Omron CX-Programmer project 新工程 (CX-Programmer 9.72)

# PLC 新PLC1: CJ1M CPU13
I/O table (CPU CJ1M-CPU13): rack 0 slot 0 CJ1W-SCU41-V1; rack 0 slot 1 CJ1W-DRM21; rack 0 slot 2 CJ1W-IA111; rack 0 slot 3 CJ1W-IA111; rack 0 slot 4 CJ1W-IA111; rack 0 slot 5 CJ1W-IA111; rack 0 slot 6 CJ1W-IA111; rack 0 slot 7 CJ1W-IA111; rack 0 slot 8 CJ1W-IA111; rack 0 slot 9 CJ1W-OC211; rack 1 slot 0 CJ1W-OC211; rack 1 slot 1 CJ1W-OC211; rack 1 slot 2 CJ1W-OC211; rack 1 slot 3 CJ1W-OC211; rack 1 slot 4 CJ1W-ID211; rack 1 slot 5 CJ1W-IA111; rack 1 slot 6 CJ1W-AD041-V1

## Global symbols (name address type ; comment)
0.00 BOOL  ; 右前按钮站闭点并
0.01 BOOL  ; 右前按钮站闭点串
0.02 BOOL  ; 右前按钮站开点串
0.04 BOOL  ; 左后按钮站闭点并
0.05 BOOL  ; 左后按钮站闭点串
0.06 BOOL  ; 左后按钮站开点串
150 CHANNEL  ; 1-16通道比较后的结果字
151 CHANNEL  ; 17-32通道比较后的结果字
2008.01 BOOL  ; RUN mode
2008.02 BOOL  ; 电子凸轮模块故障
2008.04 BOOL  ; Memory load completed
2008.06 BOOL  ; Memory load enable
30.00 BOOL  ; 高油压
30.01 BOOL  ; 1#高油压
30.03 BOOL  ; 主润滑次数正常
30.06 BOOL  ; 气垫润滑高压
30.07 BOOL  ; 油箱加热
30.08 BOOL  ; 润滑次数正常
30.09 BOOL  ; 低油压
30.13 BOOL  ; 主润滑次数正常
30.14 BOOL  ; 润滑正常
310.03 BOOL  ; 1#MB前开出停止
315.01 BOOL  ; 高油位
315.02 BOOL  ; 低油位
315.03 BOOL  ; 1#过滤器堵塞
315.04 BOOL  ; 2#过滤器堵塞
315.05 BOOL  ; 3#滤油器堵塞
315.06 BOOL  ; 高油压
315.07 BOOL  ; 低油压
316.00 BOOL  ; 模具更换
316.01 BOOL  ; 上死点300-0
316.02 BOOL  ; 数据编辑断
316.03 BOOL  ; 气垫落到底
316.06 BOOL  ; MB右开进停止
316.07 BOOL  ; 选择夹紧
316.08 BOOL  ; 选择放松
316.09 BOOL  ; MB落下（前）
316.10 BOOL  ; MB落下（后）
316.11 BOOL  ; MB夹紧压力
316.12 BOOL  ; MB放松压力
318.00 BOOL  ; 变频器正常
318.01 BOOL  ; 变频器电源合上
318.02 BOOL  ; 点动
318.03 BOOL  ; 单动
318.04 BOOL  ; 自动
318.05 BOOL  ; 安全栓复位
319.00 BOOL  ; 双阀故障
319.02 BOOL  ; 安全栓未就位
319.03 BOOL  ; 急停故障
319.04 BOOL  ; 工作台变频器正常
31.13 BOOL  ; 故障复位
31.14 BOOL  ; 急停防粘
31.15 BOOL  ; 紧急停止
320.02 BOOL  ; 润滑电机开关触点
320.04 BOOL  ; 电柜冷却开关触点
320.05 BOOL  ; 润滑电机停止
320.06 BOOL  ; 润滑电机开动
320.09 BOOL  ; 油箱加热开关触点
320.10 BOOL  ; 油箱温度正常
320.11 BOOL  ; 油箱加热停
320.12 BOOL  ; 油箱加热开
320.14 BOOL  ; 润滑电机运行
320.15 BOOL  ; 油箱加热
321.00 BOOL  ; 润滑正常
321.01 BOOL  ; 主电机温度正常
321.02 BOOL  ; 梯子限位
321.03 BOOL  ; 主电机热过载
321.04 BOOL  ; 主电机零速
321.10 BOOL  ; 主电机停止按钮
321.11 BOOL  ; 主电机启动按钮
321.12 BOOL  ; 飞轮制动限位1#
321.13 BOOL  ; 飞轮制动限位2#
321.15 BOOL  ; 主电机启动OK
322.00 BOOL  ; 主电机运行
322.10 BOOL  ; 数据编辑通/断
322.11 BOOL  ; 安全栓到位
322.13 BOOL  ; 液压保护过载
322.14 BOOL  ; 液压保护选择重调
323.01 BOOL  ; 液压保护正常
323.02 BOOL  ; 液压保护选择正常
324.00 BOOL  ; 选择滑块调整
324.01 BOOL  ; 滑块调整空开
324.02 BOOL  ; 点动/自动选择
324.03 BOOL  ; 上限位
324.04 BOOL  ; 下限位
324.05 BOOL  ; 滑块调整向上按钮
324.06 BOOL  ; 滑块调整向下按钮
324.14 BOOL  ; 滑块调整向上
324.15 BOOL  ; 滑块调整向下
327.00 BOOL  ; 选择行程
327.02 BOOL  ; 连续预置钮
327.03 BOOL  ; 离制压力
327.04 BOOL  ; 主电机选择正转
328.01 BOOL  ; 液压保护压力正常
328.02 BOOL  ; 液压保护限位
328.05 BOOL  ; 液压保护重调OK
329.00 BOOL  ; 选择气垫调整
329.01 BOOL  ; 气垫调整空开
329.02 BOOL  ; 气垫落到底
329.03 BOOL  ; 气垫上限位
329.04 BOOL  ; 气垫下限位
329.05 BOOL  ; 气垫向上按钮
329.06 BOOL  ; 气垫向下按钮
329.14 BOOL  ; 气垫调整向上
329.15 BOOL  ; 气垫调整向下
32.00 BOOL  ; 主电机开动条件
32.01 BOOL  ; 主电机开动
32.02 BOOL  ; 正转
32.03 BOOL  ; 反转
32.04 BOOL  ; 主电机运行
32.05 BOOL  ; 离合器动作
32.06 BOOL  ; 延时排气
32.08 BOOL  ; 进气条件
32.09 BOOL  ; 排气条件
32.14 BOOL  ; 设定条件
32.15 BOOL  ; 设定允许
330.00 BOOL  ; 气垫顶起旋钮
330.01 BOOL  ; 工作台开进到位
330.02 BOOL  ; 气垫低压进气阀
330.03 BOOL  ; 气垫高压进气阀
33.01 BOOL  ; 液保重调
33.02 BOOL  ; 液保过载
33.03 BOOL  ; 平衡器压力正常
33.04 BOOL  ; 液保与行程连锁
33.05 BOOL  ; 上死点校�
33.06 BOOL  ; BM
33.07 BOOL  ; TC
33.12 BOOL  ; 制动监控故障
342.00 BOOL  ; 高油压
342.08 BOOL  ; 油箱低油位
342.13 BOOL  ; 油泵电机空开QF11掉电
342.14 BOOL  ; 电柜风机空开QF18掉电
342.15 BOOL  ; 油泵运行OK
343.00 BOOL  ; 油箱加热温度开关断
343.01 BOOL  ; 油箱加热温度开关断
343.05 BOOL  ; 油箱加热OK
343.06 BOOL  ; 润滑不正常
343.07 BOOL  ; 梯子限位未复位
343.08 BOOL  ; 电机温度保护
343.09 BOOL  ; 热过载
343.11 BOOL  ; 飞轮刹车限位未接通
344.05 BOOL  ; 主电机运转条件OK
344.06 BOOL  ; SK2开关选择不正确
344.07 BOOL  ; 数据编辑未选择断
344.08 BOOL  ; 平衡器压力不正常
344.13 BOOL  ; 安全栓未复位
344.14 BOOL  ; 紧急停止未复位
344.15 BOOL  ; 故障未复位
345.00 BOOL  ; 工作台未落下夹紧
345.01 BOOL  ; 液压保护开关位置不正确
345.02 BOOL  ; 1#托板未落下
345.06 BOOL  ; 寸动运转方向选择不正确
345.07 BOOL  ; 微调刹车限位未接通
345.08 BOOL  ; 微调电机空开QF3掉电
345.15 BOOL  ; 微调OK
346.00 BOOL  ; 滑块液保不正常
346.04 BOOL  ; 自动开时设定值与实际值偏差应大于50mm
346.07 BOOL  ; 滑块调整断轴
346.10 BOOL  ; 调整到上限位
346.11 BOOL  ; 调整到下限位
346.12 BOOL  ; 滑块调整 空开QF4掉电
346.14 BOOL  ; 滑块调整OK
347.00 BOOL  ; 滑块未在上死点
347.01 BOOL  ; 气垫未落到底
347.02 BOOL  ; 气垫调整 空开QF5掉电
347.03 BOOL  ; 气垫调整断轴
347.07 BOOL  ; 气垫调整断轴
347.08 BOOL  ; 气垫调整上限位
347.09 BOOL  ; 气垫调整下限位
347.10 BOOL  ; 气垫调整OK
348.00 BOOL  ; 行程开关SK3选择不正确
348.01 BOOL  ; 离制压力不正常
348.02 BOOL  ; 电子凸轮故障
348.03 BOOL  ; 光电保护断
348.05 BOOL  ; 双阀故障
348.15 BOOL  ; 寸动OK
349.01 BOOL  ; 气垫润滑高压
349.03 BOOL  ; 主电机未运行
349.04 BOOL  ; 产品计数到
349.05 BOOL  ; 制动监控故障
349.06 BOOL  ; 装模高度当前值与行程联锁不正确
349.14 BOOL  ; 单次OK
349.15 BOOL  ; 连续OK
34.00 BOOL  ; 进气条件
34.01 BOOL  ; 排气条件
34.02 BOOL  ; 气垫压力正常
34.03 BOOL  ; 运行中正常
34.04 BOOL  ; 运行中正常
34.07 BOOL  ; 运行中正常
34.14 BOOL  ; 设定条件
34.15 BOOL  ; 设定允许
351.00 BOOL  ; SK4未选择 ”重调“
351.01 BOOL  ; 滑块液保限位不正常
351.06 BOOL  ; 滑块液保重调OK
351.07 BOOL  ; 滑块液保正常
352.00 BOOL  ; 滑块未在下死点
352.01 BOOL  ; 滑块未在上死点
352.07 BOOL  ; 模具更换OK
352.15 BOOL  ; 气垫顶起OK
353.00 BOOL  ; 1#托板顶起开关SA23未选择顶起
353.01 BOOL  ; 1#托板顶起电机空开QF9掉电
353.02 BOOL  ; 1#工作台位置不正确
353.14 BOOL  ; 1#托板顶起条件OK
35.01 BOOL  ; 闭点并
35.02 BOOL  ; 闭点串
35.03 BOOL  ; 开点串
35.06 BOOL  ; 防重复继电�
35.07 BOOL  ; 单连行程控制
35.10 BOOL  ; 寸动继电�
36.01 BOOL  ; 液保与行程联锁
37.00 BOOL  ; 紧急停止
37.01 BOOL  ; 电子凸轮故障
37.02 BOOL  ; 故障复位
37.03 BOOL  ; 托板落下联锁
37.04 BOOL  ; 模具完全夹紧或放松
37.05 BOOL  ; 滑块调整条件
37.06 BOOL  ; 传感器不动检测
37.07 BOOL  ; 滑块调整断轴
37.08 BOOL  ; 滑块调整断轴自保点
37.10 BOOL  ; 换模导轨顶起
37.14 BOOL  ; 设定条件
37.15 BOOL  ; 设定允许
40.01 BOOL  ; 上限位
40.02 BOOL  ; 下限位
40.03 BOOL  ; 启动自动调整
40.04 BOOL  ; 设定值与实际值之差小于20丝
40.05 BOOL  ; 允许向上自动开
40.06 BOOL  ; 故障提示用
40.07 BOOL  ; 实际值与设定值之差小于20丝
40.08 BOOL  ; 允许向下自动开
40.09 BOOL  ; 故障提示用
40.10 BOOL  ; 调整到位
40.11 BOOL  ; 向上超调
40.12 BOOL  ; 向下自动停
40.13 BOOL  ; 启动脉冲
41.00 BOOL  ; 启动自动脉冲
41.01 BOOL  ; 自动向上
41.02 BOOL  ; 调整到位
41.03 BOOL  ; 延时断
41.04 BOOL  ; 自动向下
41.05 BOOL  ; 滑块向上调整
41.06 BOOL  ; 滑块向下调整
41.10 BOOL  ; 装模高度与行程联锁
41.11 BOOL  ; 密码正确
41.12 BOOL  ; 是
41.14 BOOL  ; 设定条件
41.15 BOOL  ; 设定允许
42.00 BOOL  ; 气垫调整条件
42.01 BOOL  ; 触摸屏“-”号显示
42.06 BOOL  ; 传感器不动检测
42.07 BOOL  ; 气垫调整断轴
42.08 BOOL  ; 气垫调整断轴
42.14 BOOL  ; 设定条件
42.15 BOOL  ; 设定允许
45.01 BOOL  ; 上限位
45.02 BOOL  ; 下限位
45.03 BOOL  ; 启动自动调整
45.04 BOOL  ; 设定值与实际值之差小于20丝(向上到位)
45.05 BOOL  ; 允许向上自动开
45.06 BOOL  ; 故障提示用
45.07 BOOL  ; 实际值与设定值之差小于20丝(向下到位)
45.08 BOOL  ; 允许向下自动开
45.09 BOOL  ; 故障提示用
45.10 BOOL  ; 调整到位
45.11 BOOL  ; 向上自动停
45.12 BOOL  ; 向下自动停
45.13 BOOL  ; 托板落下
46.01 BOOL  ; 自动向上
46.04 BOOL  ; 自动向下
46.05 BOOL  ; 气垫向上调整
46.06 BOOL  ; 气垫向下调整
46.11 BOOL  ; 气垫高度密码正确
46.12 BOOL  ; 是
46.14 BOOL  ; 设定条件
46.15 BOOL  ; 设定允许
48.08 BOOL  ; 自动进角控制
49.00 BOOL  ; 点动控制条件
49.02 BOOL  ; 点动前开（正转）
49.03 BOOL  ; 点动后开（反转）
50.00 BOOL  ; 单动控制条件
50.02 BOOL  ; 单动前开（正转）
50.03 BOOL  ; 单动高速前开
50.04 BOOL  ; 单动低速前开
50.05 BOOL  ; 单动后开（反转）
50.06 BOOL  ; 单动高速后开
50.07 BOOL  ; 单动低速后开
51.00 BOOL  ; 模具更换条件
51.01 BOOL  ; 滑块模具放松
51.02 BOOL  ; 滑块模具夹紧
51.11 BOOL  ; 1#工作台上浮检测正常
51.12 BOOL  ; 2#工作台上浮检测正常
52.00 BOOL  ; 移动工作台开动条件1
52.02 BOOL  ; 移动工作台落下
52.03 BOOL  ; 移动工作台夹紧
52.04 BOOL  ; 工作台落下夹紧
52.05 BOOL  ; 移动工作台放松
52.06 BOOL  ; 工作台顶起到位
52.07 BOOL  ; 移动工作台顶起
600.00 BOOL  ; 连续停止角度
61.00 BOOL  ; 制动监控继电器
61.01 BOOL  ; 上电复位
61.02 BOOL  ; 上死点校正继电器
61.03 BOOL  ; 制动监控故障
61.12 BOOL  ; 单次
61.13 BOOL  ; 连续
61.14 BOOL  ; 寸动
61.15 BOOL  ; 离制压力
62.00 BOOL  ; 光电保护与行程联�
62.01 BOOL  ; 闭点并
62.02 BOOL  ; 闭点串
62.03 BOOL  ; 开点串
62.04 BOOL  ; 开动条件
62.05 BOOL  ; 单连条件
62.05 BOOL  ; 单连条件
62.06 BOOL  ; 单次条件
62.07 BOOL  ; 连续条件
62.08 BOOL  ; 单连条件
62.09 BOOL  ; 安全继电器
62.10 BOOL  ; 防重复继电器
62.11 BOOL  ; 单连行程控制
62.12 BOOL  ; 单连行程控制
62.13 BOOL  ; 寸动继电器
62.14 BOOL  ; 停上死点继电器
63.11 BOOL  ; 计数到
63.12 BOOL  ; 产品计数清零
63.13 BOOL  ; 产品计数通/断
63.14 BOOL  ; 产品计数设定条件
63.15 BOOL  ; 产品计数设定允许
64.00 BOOL  ; 设定条件
64.01 BOOL  ; 设定允许
64.02 BOOL  ; 1#使用设定条件
64.03 BOOL  ; 1#使用
64.04 BOOL  ; 2#使用设定条件
64.05 BOOL  ; 2#使用
64.06 BOOL  ; 3#使用设定条件
64.07 BOOL  ; 3#使用
64.08 BOOL  ; 4#使用设定条件
64.09 BOOL  ; 4#使用
65.06 BOOL  ; 1#通角度设定触发
65.07 BOOL  ; 2#通角度设定触发
65.08 BOOL  ; 3#通角度设定触发
65.09 BOOL  ; 4#通角度设定触发
66.02 BOOL  ; 1#延时使用条件
66.03 BOOL  ; 1#延时使用
66.04 BOOL  ; 2#延时使用条件
66.05 BOOL  ; 2#延时使用
66.06 BOOL  ; 3#延时使用条件
66.07 BOOL  ; 3#延时使用
66.08 BOOL  ; 4#延时使用条件
66.09 BOOL  ; 4#延时使用
67.06 BOOL  ; 1#延时时间设定触发
67.07 BOOL  ; 2#延时时间设定触发
67.08 BOOL  ; 3#延时时间设定触发
67.09 BOOL  ; 4#延时时间设定触发
68.06 BOOL  ; 1#断角度设定触发
68.07 BOOL  ; 2#断角度设定触发
68.08 BOOL  ; 3#断角度设定触发
68.09 BOOL  ; 4#断角度设定触发
69.03 BOOL  ; 1#气源用凸轮
69.06 BOOL  ; 2#气源用凸轮
69.09 BOOL  ; 3#气源用凸轮
69.12 BOOL  ; 4#气源用凸轮
71.01 BOOL  ; 1#气源延时起动
71.02 BOOL  ; 2#气源延时起动
71.03 BOOL  ; 3#气源延时起动
71.04 BOOL  ; 4#气源延时起动
72.00 BOOL  ; 密码正确
72.01 BOOL  ; 参数设置条件
72.02 BOOL  ; 参数设置允许
72.07 BOOL  ; 参数确认
72.08 BOOL  ; 参数确认是
72.09 BOOL  ; $?St$Bk?_#[5] / 参数设置"是"$?St$Bk?_#[5]
72.11 BOOL  ; $?St$Bk?_#[6] / 参数设置"否"$?St$Bk?_#[6]
72.15 BOOL  ; 模具号选择
73.01 BOOL  ; 模具更换选择条件
73.02 BOOL  ; 模具更换选择通
73.07 BOOL  ; 换模确认选择条件
73.08 BOOL  ; 换模确认选择通
73.09 BOOL  ; $?St$Bk?_#[7] / 参数确认"是"$?St$Bk?_#[7]
73.11 BOOL  ; 换模确认”否“
77.01 BOOL  ; 操作“+ “
77.02 BOOL  ; 操作”-“
78.01 BOOL  ; 油泵OK监控
78.02 BOOL  ; 主电机OK监控
78.03 BOOL  ; 微调OK监控
78.04 BOOL  ; 滑块调整
78.06 BOOL  ; 气垫调整
78.07 BOOL  ; 栅栏升降
78.08 BOOL  ; 寸动
78.09 BOOL  ; 单次
78.10 BOOL  ; 连续
78.12 BOOL  ; 滑块液压保护重调
78.14 BOOL  ; 气垫调整
78.15 BOOL  ; 气垫顶起
79.00 BOOL  ; 托板顶起
D15000 CHANNEL  ; 电子凸轮32通道中第1通道
D15032 CHANNEL  ; 防重复通角度[17]
D15033 CHANNEL  ; 防重复断角度[17]
D15034 CHANNEL  ; 过载重调通角度[18]
D15035 CHANNEL  ; 过载重调断角度[18]
D15036 CHANNEL  ; 微调返回通角度[19]
D15037 CHANNEL  ; 微调返回断角度[19]
D15038 CHANNEL  ; 光电保护通角度[20]
D15039 CHANNEL  ; 光电保护断角度[20]
D15040 CHANNEL  ; 产品计数通角度[21]
D15041 CHANNEL  ; 产品计数断角度[21]
D15042 CHANNEL  ; 下死点通角度[22]
D15043 CHANNEL  ; 下死点断角度[22]
D15044 CHANNEL  ; 气垫闭锁通角度[23]
D15045 CHANNEL  ; 气垫闭锁断角度[23]
D15046 CHANNEL  ; 平衡器压力进气通角度[24]
D15047 CHANNEL  ; 平衡器压力进气断角度[24]
D15048 CHANNEL  ; 平衡器压力排气通角度[25]
D15049 CHANNEL  ; 平衡器压力排气断角度[25]
D15050 CHANNEL  ; 气垫压力控制通角度[26]
D15051 CHANNEL  ; 气垫压力控制断角度[26]
D15052 CHANNEL  ; 上死点校核通角度[27]
D15053 CHANNEL  ; 上死点校核断角度[27]
D15054 CHANNEL  ; 停在上死点故障通角度[28]
D15055 CHANNEL  ; 停在上死点故障断角度[28]
D15060 CHANNEL  ; 单次返回通角度[31]
D15061 CHANNEL  ; 单次返回断角度[31]
D2001 CHANNEL  ; 1#打油次数当前值
D2003 CHANNEL  ; 3#打油次数设定值
D20100 CHANNEL  ; 模拟量输入用2个通道(0011)=3
D20101 CHANNEL  ; 模拟量2个通道代码(00001010)=A
D2021 CHANNEL  ; 主分油器次数设定值
D2022 CHANNEL  ; 连杆打油次数设定值
D2023 CHANNEL  ; 打油次数设定值
D2041 CHANNEL  ; 平衡器压力实际值
D2043 CHANNEL  ; 设-实
D2044 CHANNEL  ; 实-设
D2046 CHANNEL  ; 实际值的1.3倍
D2049 CHANNEL  ; 实际值的0.95倍
D2081 CHANNEL  ; 气垫压力实际值
D2083 CHANNEL  ; 设-实
D2084 CHANNEL  ; 实-设
D2108 CHANNEL  ; 触摸屏显示转数
D2132 CHANNEL  ; 装模高度实际值
D2134 CHANNEL  ; 设定值与实际值之差
D2136 CHANNEL  ; 实际值与设定值之差
D2138 CHANNEL  ; 实际值(BCD)
D2148 CHANNEL  ; 密码
D2150 CHANNEL  ; 触摸屏输入的当前值
D2166 CHANNEL  ; 自动测定减速距离
D2208 CHANNEL  ; 触摸屏显示转数
D2228 CHANNEL  ; 修正值
D2232 CHANNEL  ; 气垫调整实际值
D2234 CHANNEL  ; 设定值与实际值之差
D2236 CHANNEL  ; 实际值与设定值之差
D2250 CHANNEL  ; 触摸屏输入的当前值
D2400 CHANNEL  ; #8192
D2402 CHANNEL  ; X与（Y与4096的积）约分的分子
D2404 CHANNEL  ; X与（Y与8192的积）约分的分母
D2406 CHANNEL  ; 上限80000
D2408 CHANNEL  ; 下限48000
D2410 CHANNEL  ; #20
D2414 CHANNEL  ; #150
D2416 CHANNEL  ; #28
D2418 CHANNEL  ; #5000
D2420 CHANNEL  ; 8192*8192
D2422 CHANNEL  ; #50
D2426 CHANNEL  ; 软限位上限
D2428 CHANNEL  ; 软限位下限
D2434 CHANNEL  ; BCD 2mm
D2436 CHANNEL  ; BCD 0.3mm
D2500 CHANNEL  ; #8192
D2502 CHANNEL  ; 变比乘
D2504 CHANNEL  ; 变比除
D2506 CHANNEL  ; 上限20000
D2508 CHANNEL  ; 下限#0
D2510 CHANNEL  ; #20
D2514 CHANNEL  ; #50
D2516 CHANNEL  ; #50
D2518 CHANNEL  ; #5000
D2526 CHANNEL  ; 软限位上限
D2528 CHANNEL  ; 软限位下限
D3001 CHANNEL  ; 平衡器压力设定值
D3003 CHANNEL  ; 气垫压力设定值
D3004 CHANNEL  ; 装模高度设定值
D3008 CHANNEL  ; 气垫调整设定值
D3012 CHANNEL  ; 产品计数设定值
D3040 CHANNEL  ; 产品计数现行值
D3066 CHANNEL  ; 制动角
D3401 CHANNEL  ; 模具号
D3403 CHANNEL  ; 参数设定首地址
D3421 CHANNEL  ; 模具参数所需地址
D3431 CHANNEL  ; 模具参数首地址
D3501 CHANNEL  ; 当前模具号
D3503 CHANNEL  ; 参数设定首地址
D3521 CHANNEL  ; 模具参数所需地址
D3531 CHANNEL  ; 模具参数所需地址
D3591 CHANNEL  ; 当前模具号
D3901 CHANNEL  ; 操作屏代码
D3903 CHANNEL  ; 操作行号
D3911 CHANNEL  ; 提示行号
D4051 CHANNEL  ; 1# CLSC39 ON 角度设定
D4052 CHANNEL  ; 1# CLSC39 OFF 角度设定
D4053 CHANNEL  ; 2# CLSC40 ON 角度设定
D4054 CHANNEL  ; 2# CLSC40 OFF 角度设定
D4055 CHANNEL  ; 3# CLSC41 ON 角度设定
D4056 CHANNEL  ; 3# CLSC41 OFF 角度设定
D4057 CHANNEL  ; 4# CLSC42 ON 角度设定
D4058 CHANNEL  ; 4# CLSC42 OFF 角度设定
D999 CHANNEL  ; 实际角度
H1.04 BOOL  ; 离合器释放异常
H1.05 BOOL  ; 转速异常
H300.00 BOOL  ; 顶起保持
H3.00 BOOL  ; 滑块模具放松
H3.02 BOOL  ; 1#工作台在里
H4.00 BOOL  ; 工作台顶起保持
T0000 BOOL  ; 平衡器润滑阀接通时间
T0003 BOOL  ; T003
T0004 BOOL  ; T004
T0006 BOOL  ; #0600润滑检测时间
T0008 BOOL  ; 低油压延时检测
T0009 BOOL  ; 寸动双手间隔时�
T0011 BOOL  ; 单连双手间隔时�
T0012 BOOL  ; 低油压延时检测
T0013 BOOL  ; 排气延时
T0015 BOOL  ; 上电复位
T0016 BOOL  ; 转速异常检测KA16吸合0.5S
T0017 BOOL  ; 转速异常检测2S延时
T0022 BOOL  ; 单连双手间隔时�
T0023 BOOL  ; 寸动双手间隔时�
T0024 BOOL  ; 单连防粘
T0025 BOOL  ; 寸动防粘
T0030 BOOL  ; 紧急停止
T0031 BOOL  ; 到位后自动延时断
T0032 BOOL  ; 反向延时
T0053 BOOL  ; 气垫低压进气阀延时断
T0055 BOOL  ; 移动工作台落下
T0056 BOOL  ; 移动工作台夹紧
T0057 BOOL  ; 移动工作台放松
T0058 BOOL  ; 移动工作台顶起
T0061 BOOL  ; 开出精定位
T0066 BOOL  ; 开进精定位
T0120 BOOL  ; 1#延时使用时间
T0121 BOOL  ; 2#延时使用时间
T0122 BOOL  ; 3#延时使用时间
T0123 BOOL  ; 4#延时使用时间
T0140 BOOL  ; 放松压力延时
T11 CHANNEL  ; 单连双手间隔时�
T9 CHANNEL  ; 寸动双手间隔时�
BPQ 4.00 BOOL  ; 变频器正常
BT 1.08 BOOL  ; 主电机温度保护
CLSA_1 5.01 BOOL  ; 防重复260-200
CLSA_2 5.02 BOOL  ; 防重复检查300-240
CLSA_3 5.03 BOOL  ; 单次返回180-330
CLSC1 12.00 BOOL  ; 电子凸轮输入1
CLSC17 151.00 BOOL  ; 防重复检查300-240
CLSC18 151.01 BOOL  ; 上死点330-30
CLSC19 151.02 BOOL  ; 微调返回0-180
CLSC2 12.01 BOOL  ; 电子凸轮输入2
CLSC21 151.04 BOOL  ; 产品计数240-290
CLSC22 151.05 BOOL  ; 下死点175-185
CLSC24 151.07 BOOL  ; 进气角度330-30
CLSC25 151.08 BOOL  ; 排气角度185-210
CLSC26 151.09 BOOL  ; 气垫进排气角度330-30
CLSC27 151.10 BOOL  ; 上死点校核350-290
CLSC28 151.11 BOOL  ; 停在上死点故障90-30
CLSC29 151.12 BOOL  ; 备用
CLSC3 12.02 BOOL  ; 电子凸轮输入3
CLSC31 151.14 BOOL  ; 单次返回180-330
CLSC4 12.03 BOOL  ; 电子凸轮输入4
CLSC5 12.04 BOOL  ; 电子凸轮输入5
CLSC6 12.05 BOOL  ; 电子凸轮输入6
CLSC7 12.06 BOOL  ; 电子凸轮输入7
CLSC8 12.07 BOOL  ; 电子凸轮输入8
CLSC9 12.08 BOOL  ; 电子凸轮输入9
FR1 1.01 BOOL  ; 主电机热过载
HL1 7.08 BOOL  ; 主电机运行
HL11 8.03 BOOL  ; 故障
HL12 8.06 BOOL  ; 液保过载
HL13 8.07 BOOL  ; 液保正常
HL14 10.00 BOOL  ; 滤油器堵塞指示
HL15_16 8.14 BOOL  ; 移动按钮站插入
HL19 11.08 BOOL  ; 滑块模具夹紧灯
HL2 7.00 BOOL  ; PLC运行
HL20 11.09 BOOL  ; 滑块模具放松灯
HL21 9.09 BOOL  ; 工作台夹紧到位
HL22 9.11 BOOL  ; 工作台顶起到位
HL3 7.01 BOOL  ; 电池电压低
HL32 8.01 BOOL  ; 连续予置
HL4 7.03 BOOL  ; 润滑电机运行
HL49 10.02 BOOL  ; 油箱加热指示
HL5 7.06 BOOL  ; 润滑正常
HL50 10.07 BOOL  ; 夹紧油箱低油位指示
HL6 7.04 BOOL  ; 低油位
HL7 7.05 BOOL  ; 高油位
HL8 8.15 BOOL  ; 上死点
HL9 9.00 BOOL  ; 下死点
KA11 2.04 BOOL  ; 紧急停止
KA12 2.05 BOOL  ; 紧急停止
KA13 2.11 BOOL  ; 双阀故障
KA16 2.06 BOOL  ; 双阀控制反馈1#
KA16_O 7.13 BOOL  ; 离制双阀继电器1#
KA17 2.07 BOOL  ; 双阀控制反馈2#
KA17_O 7.14 BOOL  ; 离制双阀继电器2#
KA18 2.08 BOOL  ; 双阀控制反馈3#
KA18_O 7.15 BOOL  ; 离制双阀继电器3#
KA19 2.09 BOOL  ; 双阀控制反馈4#
KA19_O 8.00 BOOL  ; 离制双阀继电器4#
KA2 1.05 BOOL  ; 防逆转
KA26 9.02 BOOL  ; 工作台手动
KA27 9.03 BOOL  ; 工作台低速
KA28 9.04 BOOL  ; 工作台高速
KA29 9.05 BOOL  ; 工作台反转
KA3 7.09 BOOL  ; 主电机正转继电器
KA30 9.06 BOOL  ; 工作台正转
KA31 9.07 BOOL  ; 工作台电机制动
KA4 7.10 BOOL  ; 主电机反转继电器
KA5 7.11 BOOL  ; 主电机星型运行
KA6 7.12 BOOL  ; 主电机角型运行
KA9 6.12 BOOL  ; 安全栓
KM11 8.08 BOOL  ; 滑块调整防粘
KM11_O 3.06 BOOL  ; 滑块调整防粘
KM12 8.09 BOOL  ; 滑块调整向上
KM12KM13 3.07 BOOL  ; 滑块调整防粘
KM13 8.10 BOOL  ; 滑块调整向下
KM15 10.08 BOOL  ; 气垫调整防粘
KM15NO 6.10 BOOL  ; 气垫调整防粘
KM16 10.09 BOOL  ; 气垫调整向上
KM16KM17 6.11 BOOL  ; 气垫调整防粘
KM17 10.10 BOOL  ; 气垫调整向下
KM35 7.02 BOOL  ; 润滑电机运行
KM49 10.01 BOOL  ; 油箱加热
KM66 9.13 BOOL  ; 工作台夹紧电机
PC1 8.02 BOOL  ; 行程计数
QF11 1.00 BOOL  ; 润滑电机开关触�
QF12 5.15 BOOL  ; 油箱加热开关触点
QF18 6.01 BOOL  ; 电柜冷却开关触�
QF4 3.01 BOOL  ; 滑块调整开关触点
QF5 6.05 BOOL  ; 气垫调整开关触点
QF52 3.14 BOOL  ; 工作台夹紧开关触点
QF7 3.15 BOOL  ; 工作台电机开关
SA10 3.08 BOOL  ; 气垫升降开关
SA25 6.14 BOOL  ; 平衡器压力手动/自动
SA26 6.15 BOOL  ; 气垫压力手动/自动
SA4_1 4.01 BOOL  ; 工作台夹紧
SA4_2 4.02 BOOL  ; 工作台放松
SB10 3.03 BOOL  ; 滑块调整向下
SB11SB12NC 2.01 BOOL  ; 寸动常闭串
SB11SB12NO 2.00 BOOL  ; 寸动常开串
SB13 6.06 BOOL  ; 气垫调整向上
SB14 6.07 BOOL  ; 气垫调整向下
SB15 3.11 BOOL  ; 平衡器手动润滑
SB16 3.12 BOOL  ; 气垫手动润滑
SB17 2.03 BOOL  ; 停上死点
SB18 4.05 BOOL  ; 工作台前开
SB19 4.06 BOOL  ; 工作台后开
SB2 1.02 BOOL  ; 主电机停止
SB26 2.12 BOOL  ; 故障复位
SB3 1.03 BOOL  ; 主电机开动
SB30 2.02 BOOL  ; 连续预置
SB4 0.14 BOOL  ; 润滑电机开
SB5 0.15 BOOL  ; 润滑电机停
SB61 5.13 BOOL  ; 油箱加热启动
SB62 5.14 BOOL  ; 油箱加热停止
SB9 3.02 BOOL  ; 滑块调整向上
SF1 0.10 BOOL  ; 低油位
SF2 0.11 BOOL  ; 高油位
SF3 6.02 BOOL  ; 夹紧油箱低油位
SK11_1 4.03 BOOL  ; 工作台单动
SK11_2 4.04 BOOL  ; 工作台点动
SK13 1.04 BOOL  ; 主电机正反转
SK2_1 1.09 BOOL  ; 选择气垫调整
SK2_2 1.10 BOOL  ; 选择行程
SK2_3 1.11 BOOL  ; 选择模具更换
SK2_4 1.12 BOOL  ; 选择滑块调整
SK3_1 1.13 BOOL  ; 连续SK3
SK3_2 1.14 BOOL  ; 单次SK3
SK3_3 1.15 BOOL  ; 寸动SK3
SK4_1 2.13 BOOL  ; 液保正常SK4
SK4_2 2.14 BOOL  ; 液保重调SK4
SK6 3.10 BOOL  ; 数据编辑
SK7_1 5.07 BOOL  ; 滑块模具夹紧
SK7_2 5.08 BOOL  ; 滑块模具放松
SK9 6.04 BOOL  ; 点动/自动选择
SP1 0.12 BOOL  ; 低油压
SP11 0.08 BOOL  ; 滤油器堵塞1#
SP12 0.09 BOOL  ; 滤油器堵塞2#
SP13 5.12 BOOL  ; 滤油器堵塞3#
SP2 0.13 BOOL  ; 高油压
SP22 4.07 BOOL  ; 工作台放松压力
SP23 4.08 BOOL  ; 工作台夹紧压力
SP26 2.10 BOOL  ; 离制压力
SP51 5.09 BOOL  ; 滑块夹紧压力1#
SP52 5.10 BOOL  ; 滑块夹紧压力2#
SP9_1 2.15 BOOL  ; 液保低压力正常
SP9_2 3.00 BOOL  ; 液保高压力正常
SQ2 3.09 BOOL  ; 气垫落到底
SQ21 3.04 BOOL  ; 滑块调整上限位
SQ22 3.05 BOOL  ; 滑块调整下限位
SQ29 6.08 BOOL  ; 气垫调整上限位
SQ3 1.06 BOOL  ; 梯子限位
SQ30 6.09 BOOL  ; 气垫调整下限位
SQ4 1.07 BOOL  ; 制动限位
SQ5 6.13 BOOL  ; 飞轮制动限位2#
SQQ1 5.04 BOOL  ; 主分油器润滑检测
SQQ2 5.05 BOOL  ; 左连杆润滑检测
SQQ21 4.11 BOOL  ; 工作台落下1#
SQQ22 4.12 BOOL  ; 工作台落下2#
SQQ3 5.06 BOOL  ; 右连杆润滑检测
SQQ47 4.09 BOOL  ; 工作台顶起1#
SQQ48 4.10 BOOL  ; 工作台顶起2#
SQQ81 4.13 BOOL  ; 工作台后开进减速
SQQ82 4.14 BOOL  ; 工作台后开进定位
SQQ83 4.15 BOOL  ; 工作台前开出减速
SQQ84 5.00 BOOL  ; 工作台前开出定位
TG2 6.00 BOOL  ; 油箱加热温度开关
XS13 0.03 BOOL  ; 右前移动按钮站插�
XS15 0.07 BOOL  ; 左后移动按钮站插�
YB1 9.01 BOOL  ; 报警器
YV1 7.07 BOOL  ; 飞轮制动阀
YV11 9.12 BOOL  ; 工作台落下阀
YV12 9.08 BOOL  ; 工作台夹紧阀
YV13 9.10 BOOL  ; 工作台放松阀
YV131 9.14 BOOL  ; 气垫润滑阀2#
YV132 9.15 BOOL  ; 气垫润滑阀3#
YV14 10.05 BOOL  ; 工作台顶起阀
YV16 11.00 BOOL  ; 平衡器进气阀
YV17 11.01 BOOL  ; 平衡器排气阀
YV18 11.03 BOOL  ; 气垫进气阀
YV19 11.04 BOOL  ; 气垫排气阀
YV27 10.11 BOOL  ; 气垫低压进气阀
YV28 10.12 BOOL  ; 气垫高压进气阀
YV3 8.11 BOOL  ; 平衡器润滑阀控制
YV31 10.03 BOOL  ; 自动化气源1#
YV32 10.04 BOOL  ; 自动化气源2#
YV4 8.12 BOOL  ; 气垫润滑阀1#
YV41 11.02 BOOL  ; 平衡器手动/自动转换阀
YV42 11.05 BOOL  ; 气垫手动/自动转换阀
YV57 11.10 BOOL  ; 滑块模具夹紧阀1#
YV58 11.11 BOOL  ; 滑块模具夹紧阀2#
YV7 8.05 BOOL  ; 液保气动泵阀

## Program MainProgram (cyclic task 0)

### Section 润滑

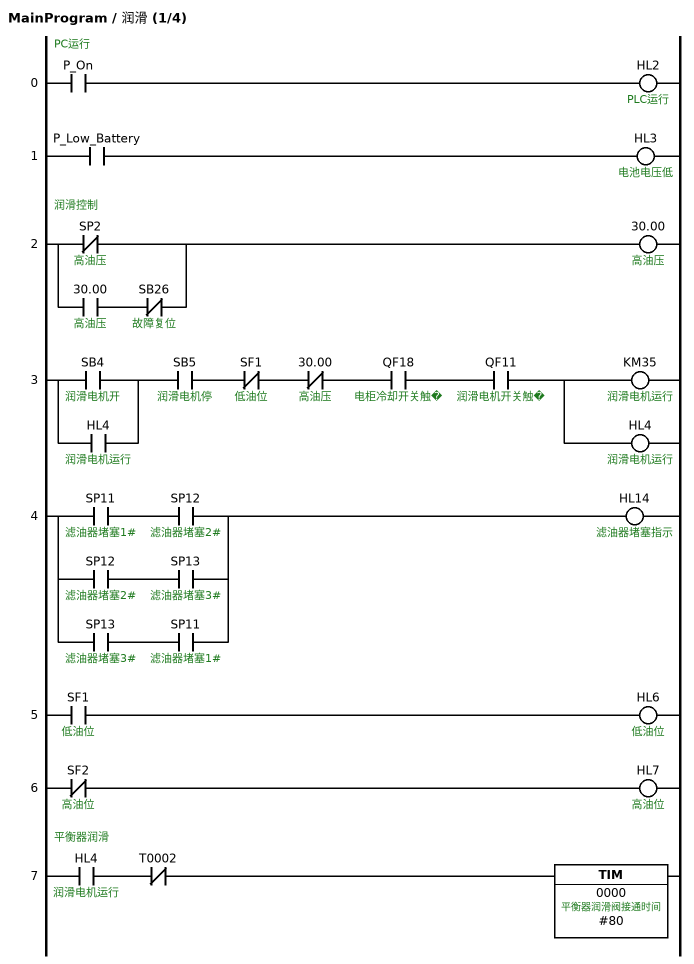
; rung 0: PC运行
LD P_On
OUT HL2  ; PLC运行
; rung 1
LD P_Low_Battery
OUT HL3  ; 电池电压低
; rung 2: 润滑控制
LDNOT SP2  ; 高油压
LD 30.00  ; 高油压
ANDNOT SB26  ; 故障复位
ORLD
OUT 30.00  ; 高油压
; rung 3
LD SB4  ; 润滑电机开
OR HL4  ; 润滑电机运行
AND SB5  ; 润滑电机停
ANDNOT SF1  ; 低油位
ANDNOT 30.00  ; 高油压
AND QF18  ; 电柜冷却开关触�
AND QF11  ; 润滑电机开关触�
OUT KM35  ; 润滑电机运行
OUT HL4  ; 润滑电机运行
; rung 4
LD SP11  ; 滤油器堵塞1#
AND SP12  ; 滤油器堵塞2#
LD SP12  ; 滤油器堵塞2#
AND SP13  ; 滤油器堵塞3#
ORLD
LD SP13  ; 滤油器堵塞3#
AND SP11  ; 滤油器堵塞1#
ORLD
OUT HL14  ; 滤油器堵塞指示
; rung 5
LD SF1  ; 低油位
OUT HL6  ; 低油位
; rung 6
LDNOT SF2  ; 高油位
OUT HL7  ; 高油位
; rung 7: 平衡器润滑
LD HL4  ; 润滑电机运行
ANDNOT T0002
TIM 0000 #80  ; 平衡器润滑阀接通时间

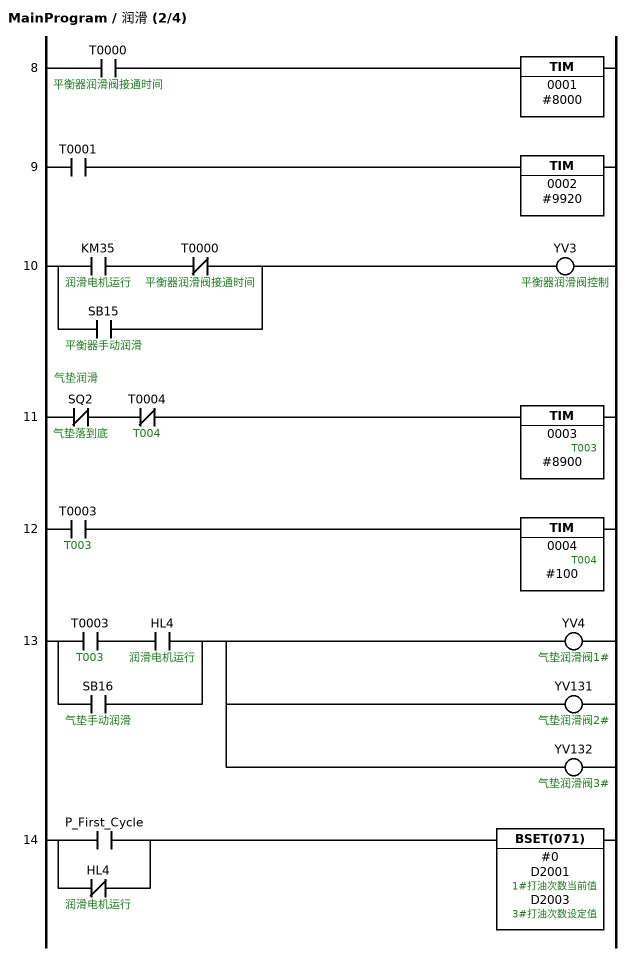
; rung 8
LD T0000  ; 平衡器润滑阀接通时间
TIM 0001 #8000
; rung 9
LD T0001
TIM 0002 #9920
; rung 10
LD KM35  ; 润滑电机运行
ANDNOT T0000  ; 平衡器润滑阀接通时间
OR SB15  ; 平衡器手动润滑
OUT YV3  ; 平衡器润滑阀控制
; rung 11: 气垫润滑
LDNOT SQ2  ; 气垫落到底
ANDNOT T0004  ; T004
TIM 0003 #8900  ; T003
; rung 12
LD T0003  ; T003
TIM 0004 #100  ; T004
; rung 13
LD T0003  ; T003
AND HL4  ; 润滑电机运行
OR SB16  ; 气垫手动润滑
OUT YV4  ; 气垫润滑阀1#
OUT YV131  ; 气垫润滑阀2#
OUT YV132  ; 气垫润滑阀3#
; rung 14
LD P_First_Cycle
ORNOT HL4  ; 润滑电机运行
BSET(071) #0 D2001 D2003  ; 1#打油次数当前值, 3#打油次数设定值

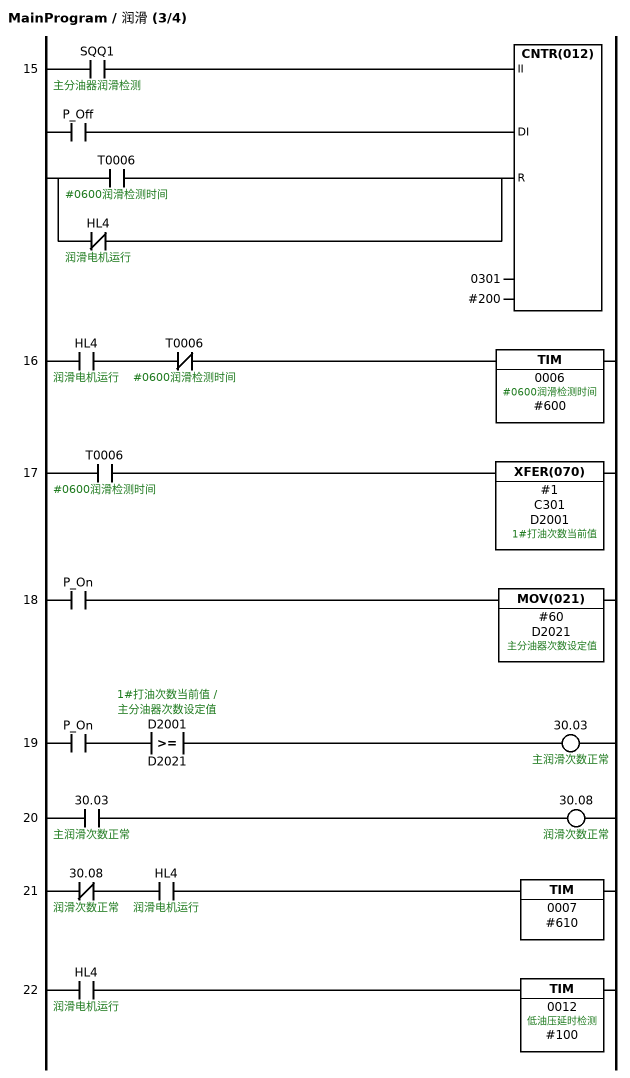
; rung 15
LD SQQ1  ; 主分油器润滑检测
LD P_Off
LD T0006  ; #0600润滑检测时间
ORNOT HL4  ; 润滑电机运行
CNTR(012) 0301 #200
; rung 16
LD HL4  ; 润滑电机运行
ANDNOT T0006  ; #0600润滑检测时间
TIM 0006 #600  ; #0600润滑检测时间
; rung 17
LD T0006  ; #0600润滑检测时间
XFER(070) #1 C301 D2001  ; 1#打油次数当前值
; rung 18
LD P_On
MOV(021) #60 D2021  ; 主分油器次数设定值
; rung 19
LD P_On
AND>=(325) D2001 D2021  ; 1#打油次数当前值, 主分油器次数设定值
OUT 30.03  ; 主润滑次数正常
; rung 20
LD 30.03  ; 主润滑次数正常
OUT 30.08  ; 润滑次数正常
; rung 21
LDNOT 30.08  ; 润滑次数正常
AND HL4  ; 润滑电机运行
TIM 0007 #610
; rung 22
LD HL4  ; 润滑电机运行
TIM 0012 #100  ; 低油压延时检测

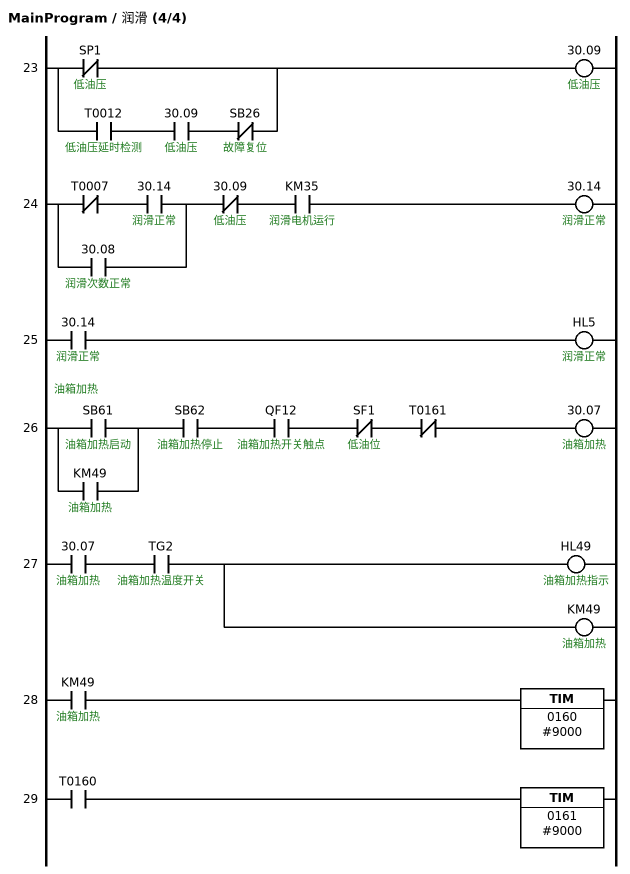
; rung 23
LDNOT SP1  ; 低油压
LD T0012  ; 低油压延时检测
AND 30.09  ; 低油压
ANDNOT SB26  ; 故障复位
ORLD
OUT 30.09  ; 低油压
; rung 24
LDNOT T0007
AND 30.14  ; 润滑正常
OR 30.08  ; 润滑次数正常
ANDNOT 30.09  ; 低油压
AND KM35  ; 润滑电机运行
OUT 30.14  ; 润滑正常
; rung 25
LD 30.14  ; 润滑正常
OUT HL5  ; 润滑正常
; rung 26: 油箱加热
LD SB61  ; 油箱加热启动
OR KM49  ; 油箱加热
AND SB62  ; 油箱加热停止
AND QF12  ; 油箱加热开关触点
ANDNOT SF1  ; 低油位
ANDNOT T0161
OUT 30.07  ; 油箱加热
; rung 27
LD 30.07  ; 油箱加热
AND TG2  ; 油箱加热温度开关
OUT HL49  ; 油箱加热指示
OUT KM49  ; 油箱加热
; rung 28
LD KM49  ; 油箱加热
TIM 0160 #9000
; rung 29
LD T0160
TIM 0161 #9000

### Section 主电机

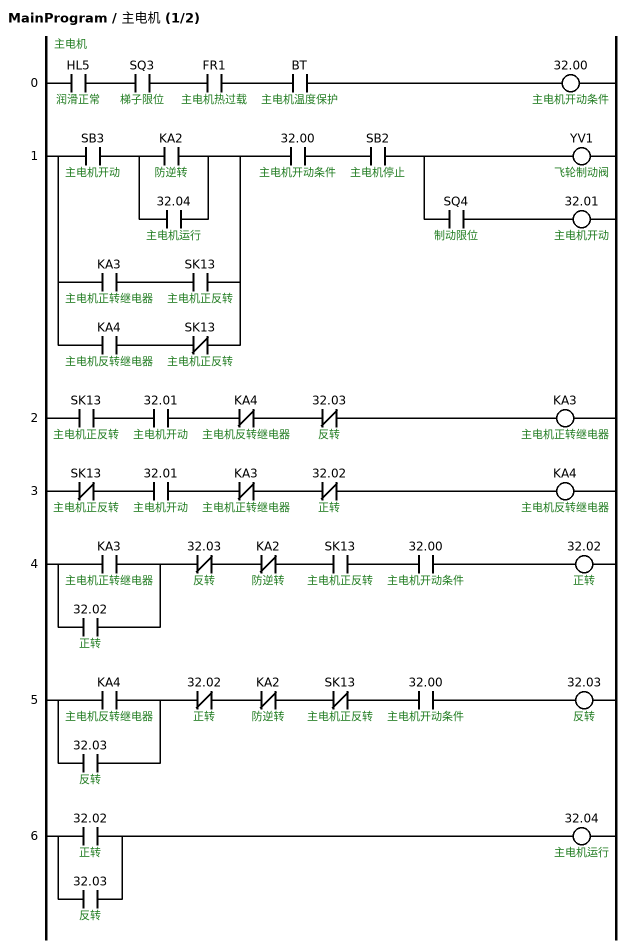
; rung 0: 主电机
LD HL5  ; 润滑正常
AND SQ3  ; 梯子限位
AND FR1  ; 主电机热过载
AND BT  ; 主电机温度保护
OUT 32.00  ; 主电机开动条件
; rung 1
LD SB3  ; 主电机开动
LD KA2  ; 防逆转
OR 32.04  ; 主电机运行
ANDLD
LD KA3  ; 主电机正转继电器
AND SK13  ; 主电机正反转
ORLD
LD KA4  ; 主电机反转继电器
ANDNOT SK13  ; 主电机正反转
ORLD
AND 32.00  ; 主电机开动条件
AND SB2  ; 主电机停止
OUT YV1  ; 飞轮制动阀
AND SQ4  ; 制动限位
OUT 32.01  ; 主电机开动
; rung 2
LD SK13  ; 主电机正反转
AND 32.01  ; 主电机开动
ANDNOT KA4  ; 主电机反转继电器
ANDNOT 32.03  ; 反转
OUT KA3  ; 主电机正转继电器
; rung 3
LDNOT SK13  ; 主电机正反转
AND 32.01  ; 主电机开动
ANDNOT KA3  ; 主电机正转继电器
ANDNOT 32.02  ; 正转
OUT KA4  ; 主电机反转继电器
; rung 4
LD KA3  ; 主电机正转继电器
OR 32.02  ; 正转
ANDNOT 32.03  ; 反转
ANDNOT KA2  ; 防逆转
AND SK13  ; 主电机正反转
AND 32.00  ; 主电机开动条件
OUT 32.02  ; 正转
; rung 5
LD KA4  ; 主电机反转继电器
OR 32.03  ; 反转
ANDNOT 32.02  ; 正转
ANDNOT KA2  ; 防逆转
ANDNOT SK13  ; 主电机正反转
AND 32.00  ; 主电机开动条件
OUT 32.03  ; 反转
; rung 6
LD 32.02  ; 正转
OR 32.03  ; 反转
OUT 32.04  ; 主电机运行

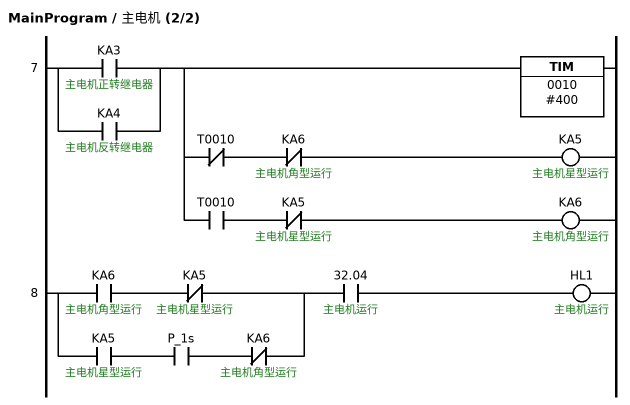
; rung 7
LD KA3  ; 主电机正转继电器
OR KA4  ; 主电机反转继电器
OUT TR0
TIM 0010 #400
ANDNOT T0010
ANDNOT KA6  ; 主电机角型运行
OUT KA5  ; 主电机星型运行
LD TR0
AND T0010
ANDNOT KA5  ; 主电机星型运行
OUT KA6  ; 主电机角型运行
; rung 8
LD KA6  ; 主电机角型运行
ANDNOT KA5  ; 主电机星型运行
LD KA5  ; 主电机星型运行
AND P_1s
ANDNOT KA6  ; 主电机角型运行
ORLD
AND 32.04  ; 主电机运行
OUT HL1  ; 主电机运行

### Section 电子凸轮

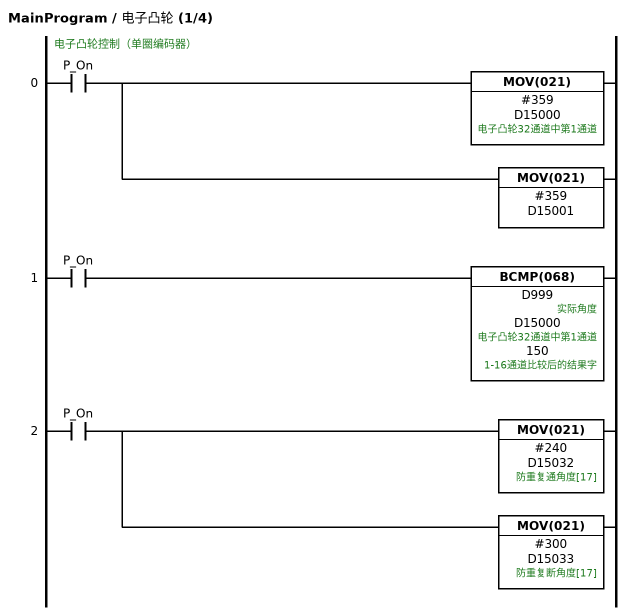
; rung 0: 电子凸轮控制（单圈编码器）
LD P_On
MOV(021) #359 D15000  ; 电子凸轮32通道中第1通道
MOV(021) #359 D15001
; rung 1
LD P_On
BCMP(068) D999 D15000 150  ; 实际角度, 电子凸轮32通道中第1通道, 1-16通道比较后的结果字
; rung 2
LD P_On
MOV(021) #240 D15032  ; 防重复通角度[17]
MOV(021) #300 D15033  ; 防重复断角度[17]

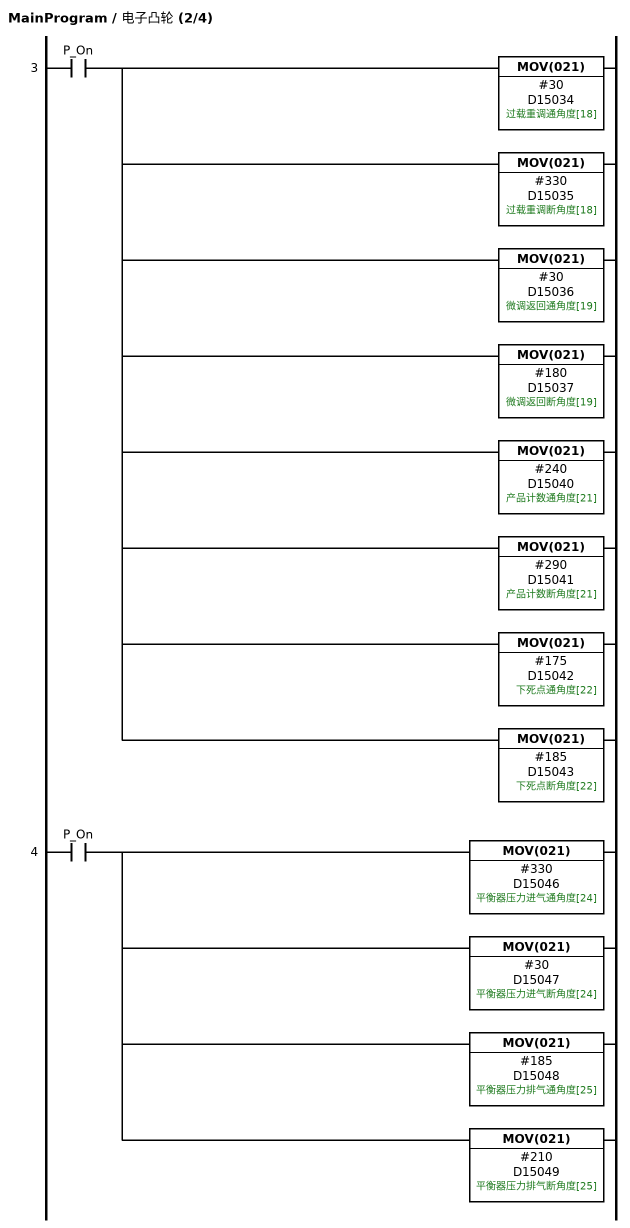
; rung 3
LD P_On
MOV(021) #30 D15034  ; 过载重调通角度[18]
MOV(021) #330 D15035  ; 过载重调断角度[18]
MOV(021) #30 D15036  ; 微调返回通角度[19]
MOV(021) #180 D15037  ; 微调返回断角度[19]
MOV(021) #240 D15040  ; 产品计数通角度[21]
MOV(021) #290 D15041  ; 产品计数断角度[21]
MOV(021) #175 D15042  ; 下死点通角度[22]
MOV(021) #185 D15043  ; 下死点断角度[22]
; rung 4
LD P_On
MOV(021) #330 D15046  ; 平衡器压力进气通角度[24]
MOV(021) #30 D15047  ; 平衡器压力进气断角度[24]
MOV(021) #185 D15048  ; 平衡器压力排气通角度[25]
MOV(021) #210 D15049  ; 平衡器压力排气断角度[25]

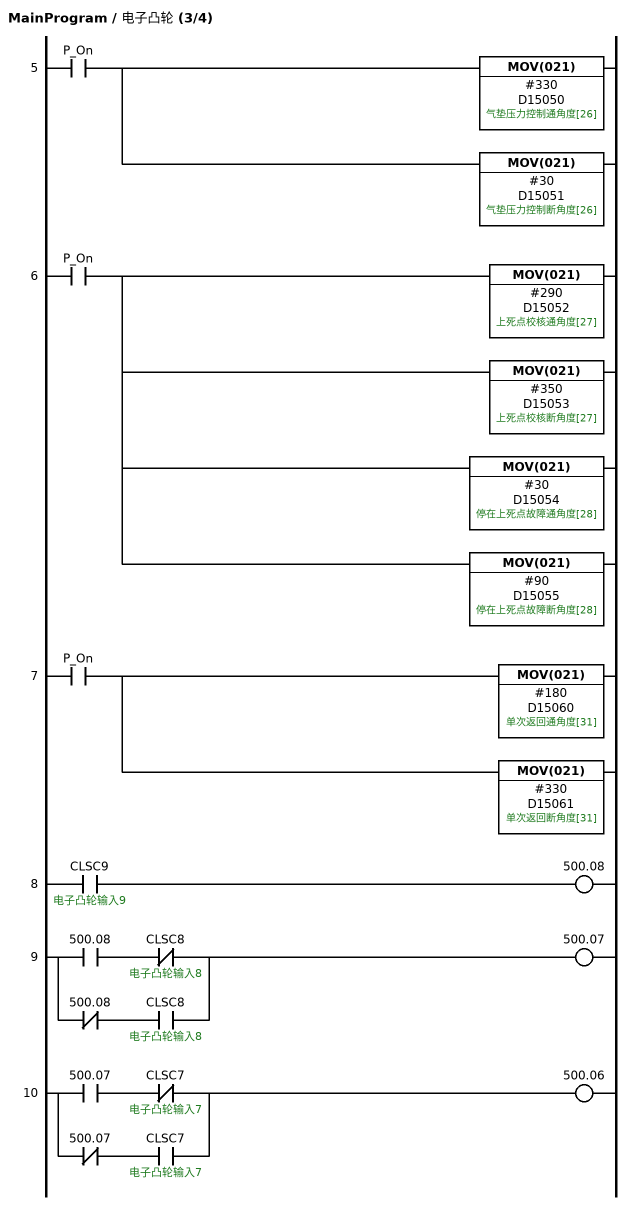
; rung 5
LD P_On
MOV(021) #330 D15050  ; 气垫压力控制通角度[26]
MOV(021) #30 D15051  ; 气垫压力控制断角度[26]
; rung 6
LD P_On
MOV(021) #290 D15052  ; 上死点校核通角度[27]
MOV(021) #350 D15053  ; 上死点校核断角度[27]
MOV(021) #30 D15054  ; 停在上死点故障通角度[28]
MOV(021) #90 D15055  ; 停在上死点故障断角度[28]
; rung 7
LD P_On
MOV(021) #180 D15060  ; 单次返回通角度[31]
MOV(021) #330 D15061  ; 单次返回断角度[31]
; rung 8
LD CLSC9  ; 电子凸轮输入9
OUT 500.08
; rung 9
LD 500.08
ANDNOT CLSC8  ; 电子凸轮输入8
LDNOT 500.08
AND CLSC8  ; 电子凸轮输入8
ORLD
OUT 500.07
; rung 10
LD 500.07
ANDNOT CLSC7  ; 电子凸轮输入7
LDNOT 500.07
AND CLSC7  ; 电子凸轮输入7
ORLD
OUT 500.06

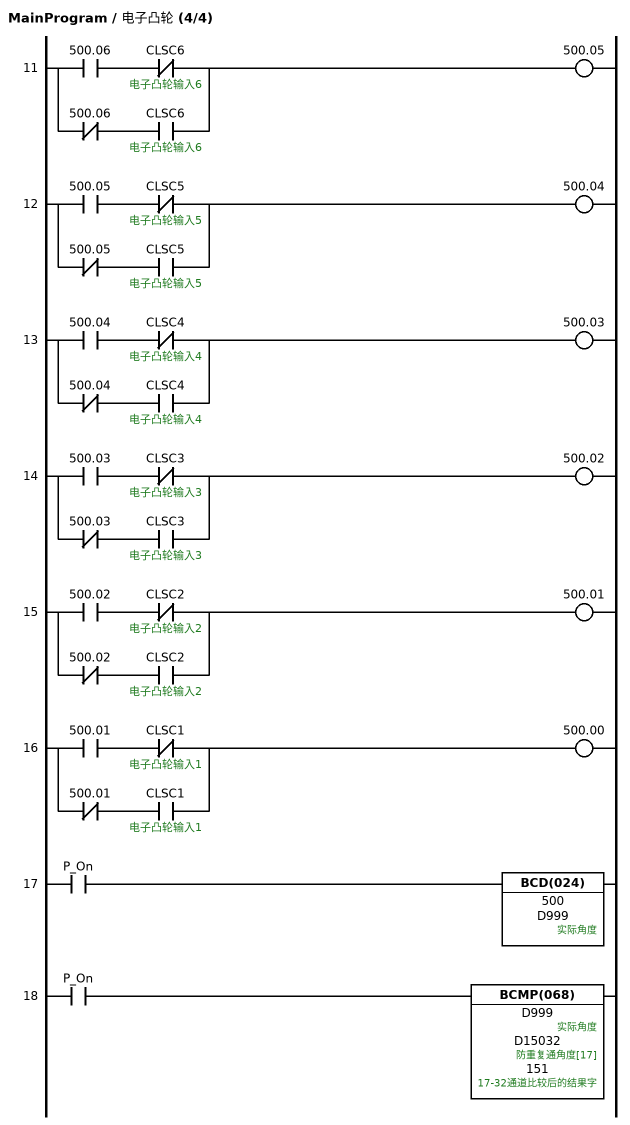
; rung 11
LD 500.06
ANDNOT CLSC6  ; 电子凸轮输入6
LDNOT 500.06
AND CLSC6  ; 电子凸轮输入6
ORLD
OUT 500.05
; rung 12
LD 500.05
ANDNOT CLSC5  ; 电子凸轮输入5
LDNOT 500.05
AND CLSC5  ; 电子凸轮输入5
ORLD
OUT 500.04
; rung 13
LD 500.04
ANDNOT CLSC4  ; 电子凸轮输入4
LDNOT 500.04
AND CLSC4  ; 电子凸轮输入4
ORLD
OUT 500.03
; rung 14
LD 500.03
ANDNOT CLSC3  ; 电子凸轮输入3
LDNOT 500.03
AND CLSC3  ; 电子凸轮输入3
ORLD
OUT 500.02
; rung 15
LD 500.02
ANDNOT CLSC2  ; 电子凸轮输入2
LDNOT 500.02
AND CLSC2  ; 电子凸轮输入2
ORLD
OUT 500.01
; rung 16
LD 500.01
ANDNOT CLSC1  ; 电子凸轮输入1
LDNOT 500.01
AND CLSC1  ; 电子凸轮输入1
ORLD
OUT 500.00
; rung 17
LD P_On
BCD(024) 500 D999  ; 实际角度
; rung 18
LD P_On
BCMP(068) D999 D15032 151  ; 实际角度, 防重复通角度[17], 17-32通道比较后的结果字

### Section 风压自动调整

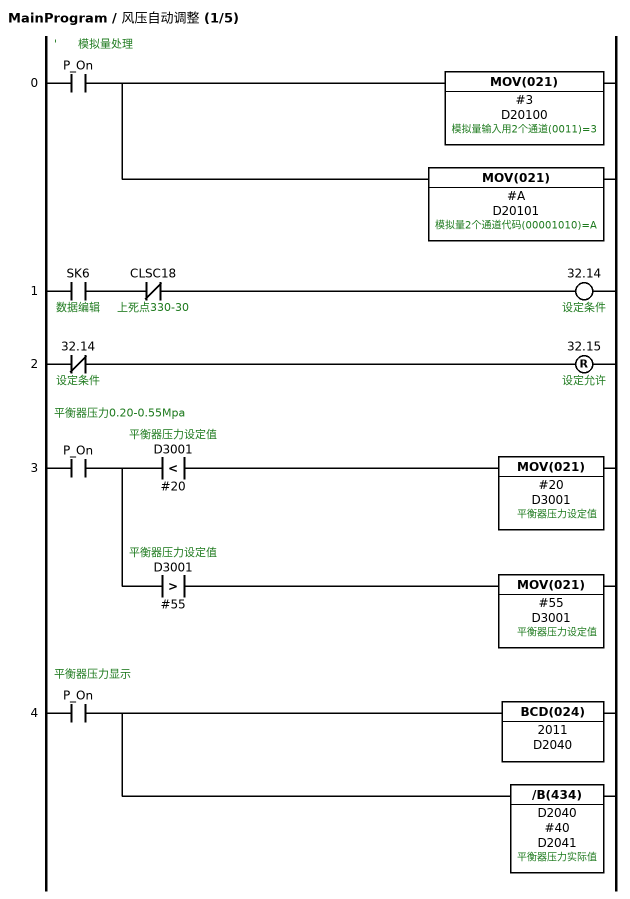
; rung 0: '      模拟量处理
LD P_On
MOV(021) #3 D20100  ; 模拟量输入用2个通道(0011)=3
MOV(021) #A D20101  ; 模拟量2个通道代码(00001010)=A
; rung 1
LD SK6  ; 数据编辑
ANDNOT CLSC18  ; 上死点330-30
OUT 32.14  ; 设定条件
; rung 2
LDNOT 32.14  ; 设定条件
RSET 32.15  ; 设定允许
; rung 3: 平衡器压力0.20-0.55Mpa
LD P_On
OUT TR0
AND<(310) D3001 #20  ; 平衡器压力设定值
MOV(021) #20 D3001  ; 平衡器压力设定值
LD TR0
AND>(320) D3001 #55  ; 平衡器压力设定值
MOV(021) #55 D3001  ; 平衡器压力设定值
; rung 4: 平衡器压力显示
LD P_On
BCD(024) 2011 D2040
/B(434) D2040 #40 D2041  ; 平衡器压力实际值

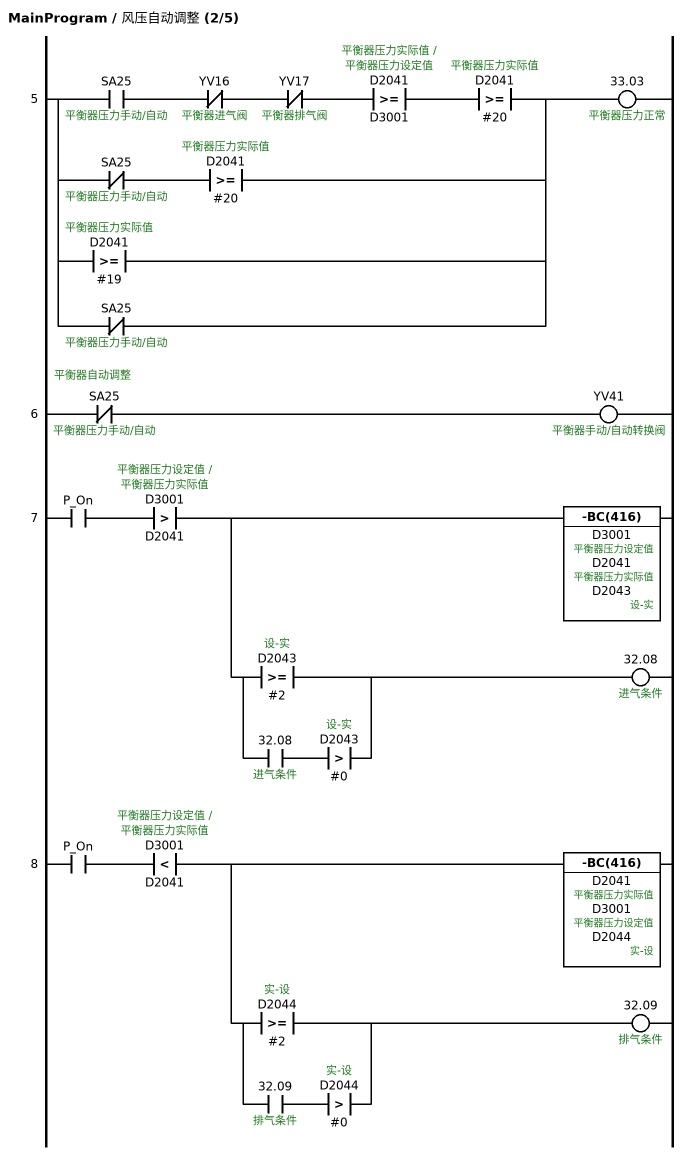
; rung 5
LD SA25  ; 平衡器压力手动/自动
ANDNOT YV16  ; 平衡器进气阀
ANDNOT YV17  ; 平衡器排气阀
AND>=(325) D2041 D3001  ; 平衡器压力实际值, 平衡器压力设定值
AND>=(325) D2041 #20  ; 平衡器压力实际值
LDNOT SA25  ; 平衡器压力手动/自动
AND>=(325) D2041 #20  ; 平衡器压力实际值
ORLD
OR>=(325) D2041 #19  ; 平衡器压力实际值
ORNOT SA25  ; 平衡器压力手动/自动
OUT 33.03  ; 平衡器压力正常
; rung 6: 平衡器自动调整
LDNOT SA25  ; 平衡器压力手动/自动
OUT YV41  ; 平衡器手动/自动转换阀
; rung 7
LD P_On
AND>(320) D3001 D2041  ; 平衡器压力设定值, 平衡器压力实际值
-BC(416) D3001 D2041 D2043  ; 平衡器压力设定值, 平衡器压力实际值, 设-实
LD>=(325) D2043 #2  ; 设-实
LD 32.08  ; 进气条件
AND>(320) D2043 #0  ; 设-实
ORLD
ANDLD
OUT 32.08  ; 进气条件
; rung 8
LD P_On
AND<(310) D3001 D2041  ; 平衡器压力设定值, 平衡器压力实际值
-BC(416) D2041 D3001 D2044  ; 平衡器压力实际值, 平衡器压力设定值, 实-设
LD>=(325) D2044 #2  ; 实-设
LD 32.09  ; 排气条件
AND>(320) D2044 #0  ; 实-设
ORLD
ANDLD
OUT 32.09  ; 排气条件

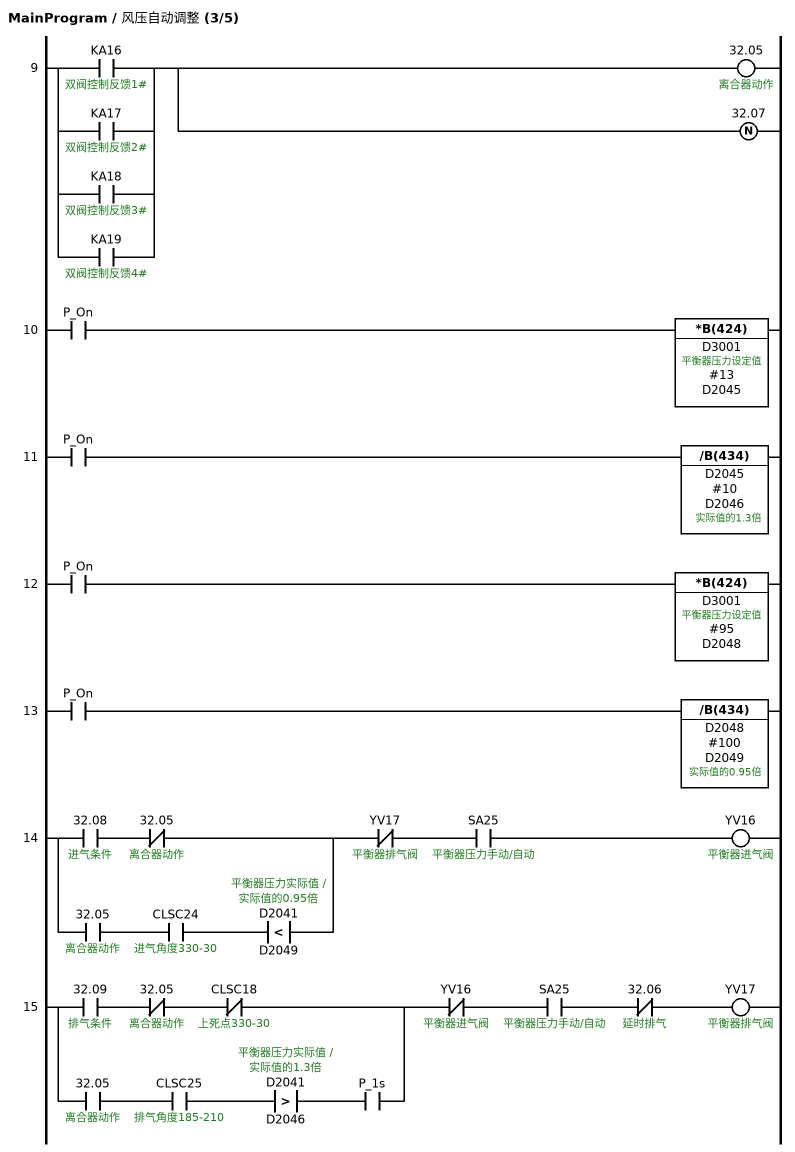
; rung 9
LD KA16  ; 双阀控制反馈1#
OR KA17  ; 双阀控制反馈2#
OR KA18  ; 双阀控制反馈3#
OR KA19  ; 双阀控制反馈4#
OUT 32.05  ; 离合器动作
DIFD(014) 32.07
; rung 10
LD P_On
*B(424) D3001 #13 D2045  ; 平衡器压力设定值
; rung 11
LD P_On
/B(434) D2045 #10 D2046  ; 实际值的1.3倍
; rung 12
LD P_On
*B(424) D3001 #95 D2048  ; 平衡器压力设定值
; rung 13
LD P_On
/B(434) D2048 #100 D2049  ; 实际值的0.95倍
; rung 14
LD 32.08  ; 进气条件
ANDNOT 32.05  ; 离合器动作
LD 32.05  ; 离合器动作
AND CLSC24  ; 进气角度330-30
AND<(310) D2041 D2049  ; 平衡器压力实际值, 实际值的0.95倍
ORLD
ANDNOT YV17  ; 平衡器排气阀
AND SA25  ; 平衡器压力手动/自动
OUT YV16  ; 平衡器进气阀
; rung 15
LD 32.09  ; 排气条件
ANDNOT 32.05  ; 离合器动作
ANDNOT CLSC18  ; 上死点330-30
LD 32.05  ; 离合器动作
AND CLSC25  ; 排气角度185-210
AND>(320) D2041 D2046  ; 平衡器压力实际值, 实际值的1.3倍
AND P_1s
ORLD
ANDNOT YV16  ; 平衡器进气阀
AND SA25  ; 平衡器压力手动/自动
ANDNOT 32.06  ; 延时排气
OUT YV17  ; 平衡器排气阀

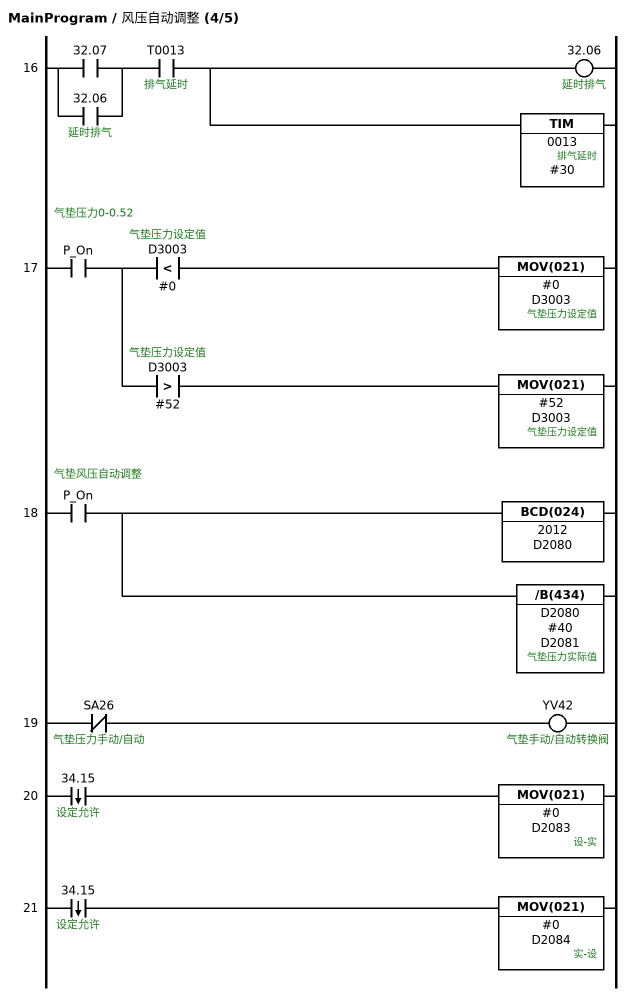
; rung 16
LD 32.07
OR 32.06  ; 延时排气
AND T0013  ; 排气延时
OUT 32.06  ; 延时排气
TIM 0013 #30  ; 排气延时
; rung 17: 气垫压力0-0.52
LD P_On
OUT TR0
AND<(310) D3003 #0  ; 气垫压力设定值
MOV(021) #0 D3003  ; 气垫压力设定值
LD TR0
AND>(320) D3003 #52  ; 气垫压力设定值
MOV(021) #52 D3003  ; 气垫压力设定值
; rung 18: 气垫风压自动调整
LD P_On
BCD(024) 2012 D2080
/B(434) D2080 #40 D2081  ; 气垫压力实际值
; rung 19
LDNOT SA26  ; 气垫压力手动/自动
OUT YV42  ; 气垫手动/自动转换阀
; rung 20
%LD 34.15  ; 设定允许
MOV(021) #0 D2083  ; 设-实
; rung 21
%LD 34.15  ; 设定允许
MOV(021) #0 D2084  ; 实-设

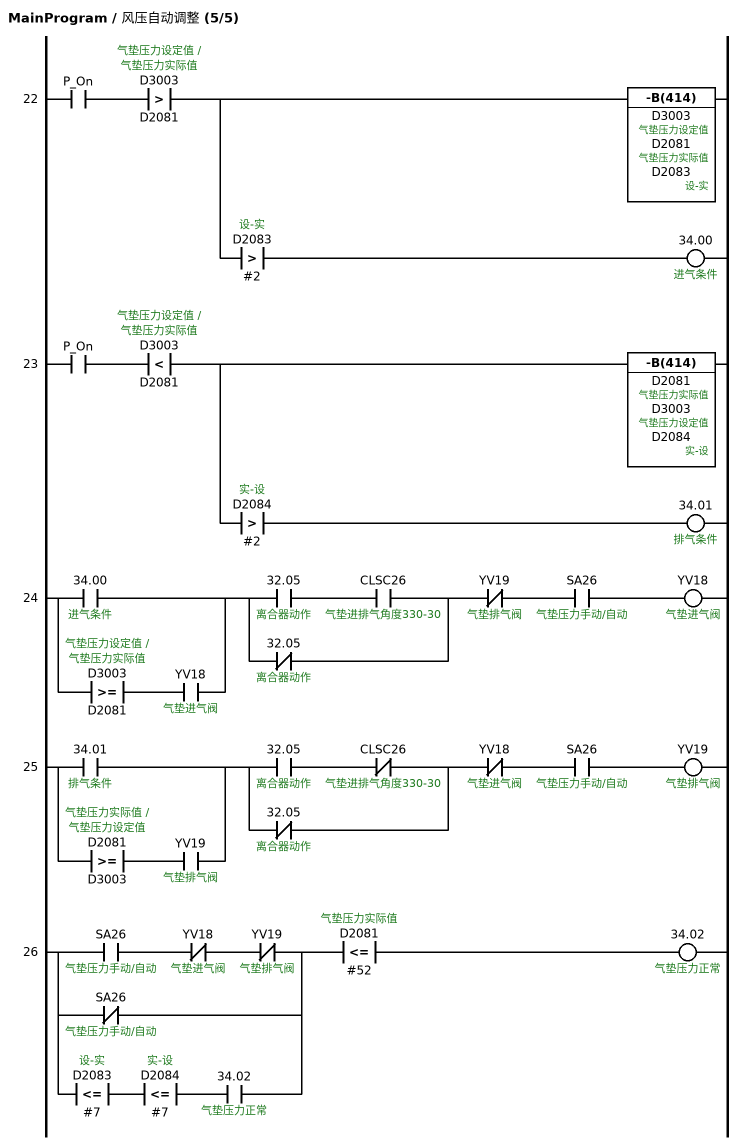
; rung 22
LD P_On
AND>(320) D3003 D2081  ; 气垫压力设定值, 气垫压力实际值
-B(414) D3003 D2081 D2083  ; 气垫压力设定值, 气垫压力实际值, 设-实
AND>(320) D2083 #2  ; 设-实
OUT 34.00  ; 进气条件
; rung 23
LD P_On
AND<(310) D3003 D2081  ; 气垫压力设定值, 气垫压力实际值
-B(414) D2081 D3003 D2084  ; 气垫压力实际值, 气垫压力设定值, 实-设
AND>(320) D2084 #2  ; 实-设
OUT 34.01  ; 排气条件
; rung 24
LD 34.00  ; 进气条件
LD>=(325) D3003 D2081  ; 气垫压力设定值, 气垫压力实际值
AND YV18  ; 气垫进气阀
ORLD
LD 32.05  ; 离合器动作
AND CLSC26  ; 气垫进排气角度330-30
ORNOT 32.05  ; 离合器动作
ANDLD
ANDNOT YV19  ; 气垫排气阀
AND SA26  ; 气垫压力手动/自动
OUT YV18  ; 气垫进气阀
; rung 25
LD 34.01  ; 排气条件
LD>=(325) D2081 D3003  ; 气垫压力实际值, 气垫压力设定值
AND YV19  ; 气垫排气阀
ORLD
LD 32.05  ; 离合器动作
ANDNOT CLSC26  ; 气垫进排气角度330-30
ORNOT 32.05  ; 离合器动作
ANDLD
ANDNOT YV18  ; 气垫进气阀
AND SA26  ; 气垫压力手动/自动
OUT YV19  ; 气垫排气阀
; rung 26
LD SA26  ; 气垫压力手动/自动
ANDNOT YV18  ; 气垫进气阀
ANDNOT YV19  ; 气垫排气阀
ORNOT SA26  ; 气垫压力手动/自动
LD<=(315) D2083 #7  ; 设-实
AND<=(315) D2084 #7  ; 实-设
AND 34.02  ; 气垫压力正常
ORLD
AND<=(315) D2081 #52  ; 气垫压力实际值
OUT 34.02  ; 气垫压力正常

### Section 液压保护

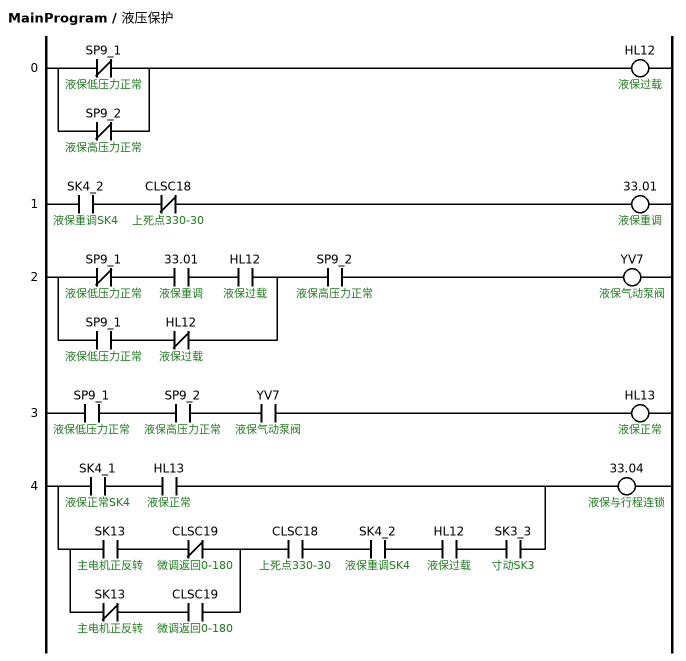
; rung 0
LDNOT SP9_1  ; 液保低压力正常
ORNOT SP9_2  ; 液保高压力正常
OUT HL12  ; 液保过载
; rung 1
LD SK4_2  ; 液保重调SK4
ANDNOT CLSC18  ; 上死点330-30
OUT 33.01  ; 液保重调
; rung 2
LDNOT SP9_1  ; 液保低压力正常
AND 33.01  ; 液保重调
AND HL12  ; 液保过载
LD SP9_1  ; 液保低压力正常
ANDNOT HL12  ; 液保过载
ORLD
AND SP9_2  ; 液保高压力正常
OUT YV7  ; 液保气动泵阀
; rung 3
LD SP9_1  ; 液保低压力正常
AND SP9_2  ; 液保高压力正常
AND YV7  ; 液保气动泵阀
OUT HL13  ; 液保正常
; rung 4
LD SK4_1  ; 液保正常SK4
AND HL13  ; 液保正常
LD SK13  ; 主电机正反转
ANDNOT CLSC19  ; 微调返回0-180
LDNOT SK13  ; 主电机正反转
AND CLSC19  ; 微调返回0-180
ORLD
AND CLSC18  ; 上死点330-30
AND SK4_2  ; 液保重调SK4
AND HL12  ; 液保过载
AND SK3_3  ; 寸动SK3
ORLD
OUT 33.04  ; 液保与行程连锁

### Section 行程

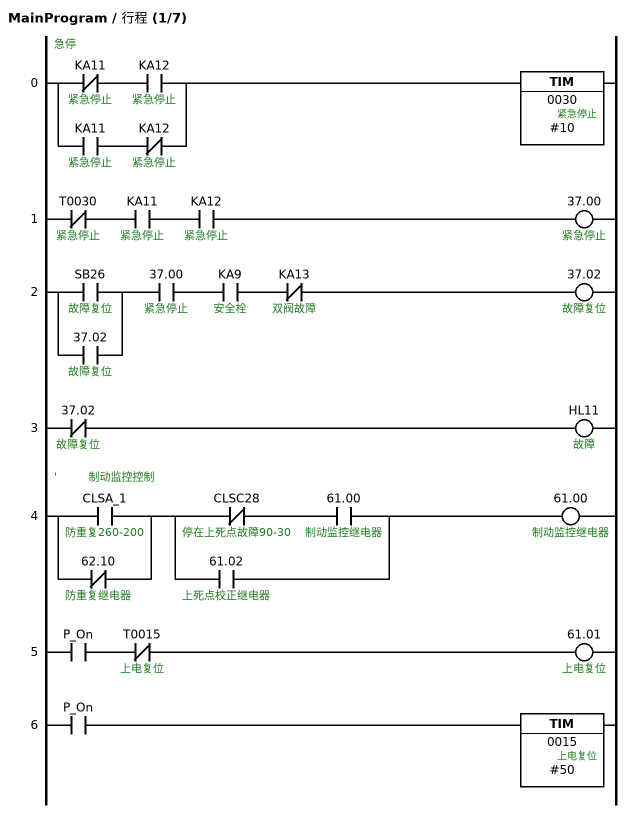
; rung 0: 急停
LDNOT KA11  ; 紧急停止
AND KA12  ; 紧急停止
LD KA11  ; 紧急停止
ANDNOT KA12  ; 紧急停止
ORLD
TIM 0030 #10  ; 紧急停止
; rung 1
LDNOT T0030  ; 紧急停止
AND KA11  ; 紧急停止
AND KA12  ; 紧急停止
OUT 37.00  ; 紧急停止
; rung 2
LD SB26  ; 故障复位
OR 37.02  ; 故障复位
AND 37.00  ; 紧急停止
AND KA9  ; 安全栓
ANDNOT KA13  ; 双阀故障
OUT 37.02  ; 故障复位
; rung 3
LDNOT 37.02  ; 故障复位
OUT HL11  ; 故障
; rung 4: '         制动监控控制
LD CLSA_1  ; 防重复260-200
ORNOT 62.10  ; 防重复继电器
LDNOT CLSC28  ; 停在上死点故障90-30
AND 61.00  ; 制动监控继电器
OR 61.02  ; 上死点校正继电器
ANDLD
OUT 61.00  ; 制动监控继电器
; rung 5
LD P_On
ANDNOT T0015  ; 上电复位
OUT 61.01  ; 上电复位
; rung 6
LD P_On
TIM 0015 #50  ; 上电复位

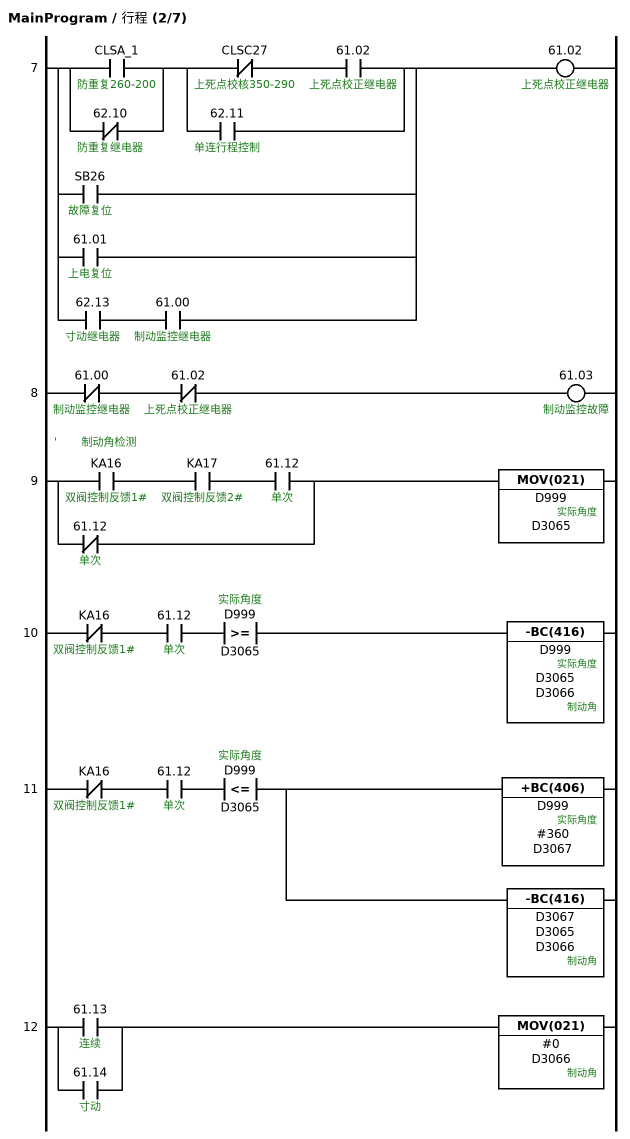
; rung 7
LD CLSA_1  ; 防重复260-200
ORNOT 62.10  ; 防重复继电器
LDNOT CLSC27  ; 上死点校核350-290
AND 61.02  ; 上死点校正继电器
OR 62.11  ; 单连行程控制
ANDLD
OR SB26  ; 故障复位
OR 61.01  ; 上电复位
LD 62.13  ; 寸动继电器
AND 61.00  ; 制动监控继电器
ORLD
OUT 61.02  ; 上死点校正继电器
; rung 8
LDNOT 61.00  ; 制动监控继电器
ANDNOT 61.02  ; 上死点校正继电器
OUT 61.03  ; 制动监控故障
; rung 9: '       制动角检测
LD KA16  ; 双阀控制反馈1#
AND KA17  ; 双阀控制反馈2#
AND 61.12  ; 单次
ORNOT 61.12  ; 单次
MOV(021) D999 D3065  ; 实际角度
; rung 10
LDNOT KA16  ; 双阀控制反馈1#
AND 61.12  ; 单次
AND>=(325) D999 D3065  ; 实际角度
-BC(416) D999 D3065 D3066  ; 实际角度, 制动角
; rung 11
LDNOT KA16  ; 双阀控制反馈1#
AND 61.12  ; 单次
AND<=(315) D999 D3065  ; 实际角度
+BC(406) D999 #360 D3067  ; 实际角度
-BC(416) D3067 D3065 D3066  ; 制动角
; rung 12
LD 61.13  ; 连续
OR 61.14  ; 寸动
MOV(021) #0 D3066  ; 制动角

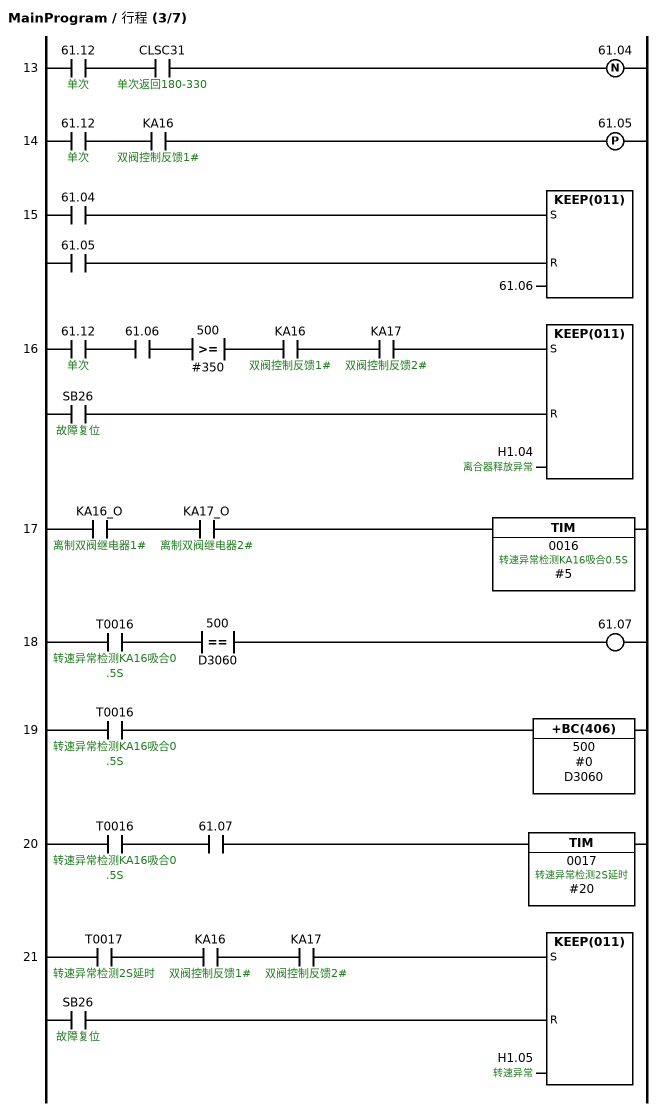
; rung 13
LD 61.12  ; 单次
AND CLSC31  ; 单次返回180-330
DIFD(014) 61.04
; rung 14
LD 61.12  ; 单次
AND KA16  ; 双阀控制反馈1#
DIFU(013) 61.05
; rung 15
LD 61.04
LD 61.05
KEEP(011) 61.06
; rung 16
LD 61.12  ; 单次
AND 61.06
AND>=(325) 500 #350
AND KA16  ; 双阀控制反馈1#
AND KA17  ; 双阀控制反馈2#
LD SB26  ; 故障复位
KEEP(011) H1.04  ; 离合器释放异常
; rung 17
LD KA16_O  ; 离制双阀继电器1#
AND KA17_O  ; 离制双阀继电器2#
TIM 0016 #5  ; 转速异常检测KA16吸合0.5S
; rung 18
LD T0016  ; 转速异常检测KA16吸合0.5S
AND=(300) 500 D3060
OUT 61.07
; rung 19
LD T0016  ; 转速异常检测KA16吸合0.5S
+BC(406) 500 #0 D3060
; rung 20
LD T0016  ; 转速异常检测KA16吸合0.5S
AND 61.07
TIM 0017 #20  ; 转速异常检测2S延时
; rung 21
LD T0017  ; 转速异常检测2S延时
AND KA16  ; 双阀控制反馈1#
AND KA17  ; 双阀控制反馈2#
LD SB26  ; 故障复位
KEEP(011) H1.05  ; 转速异常

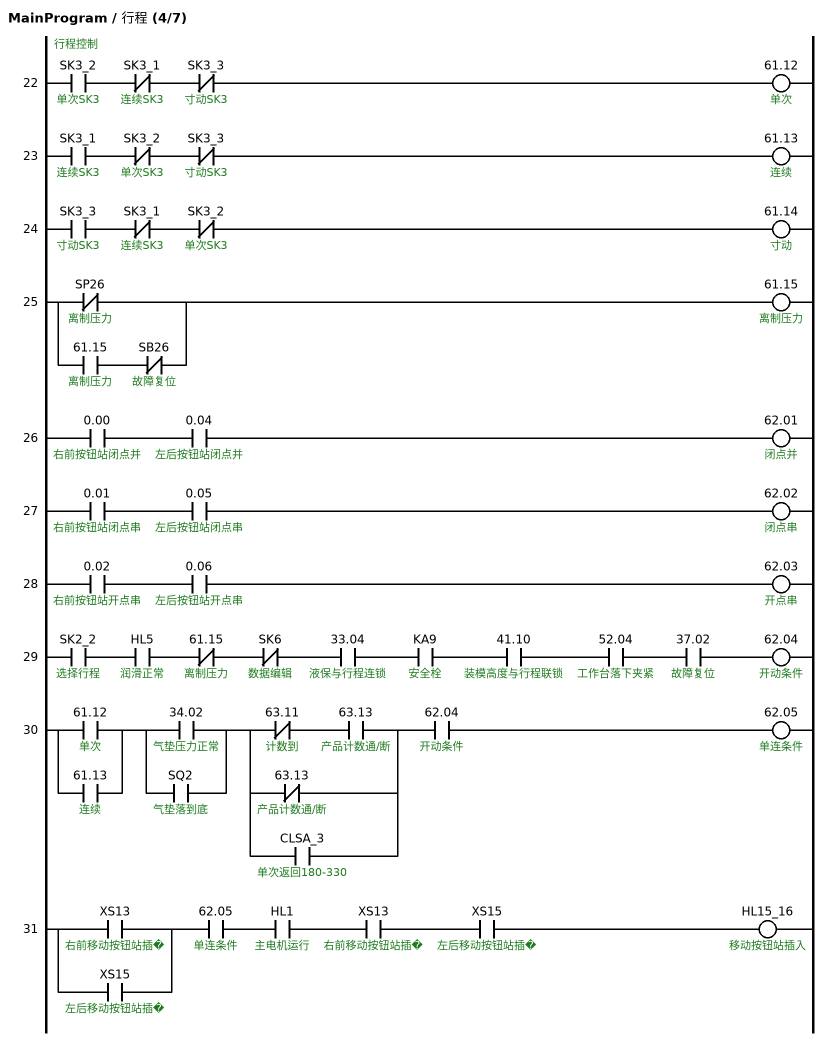
; rung 22: 行程控制
LD SK3_2  ; 单次SK3
ANDNOT SK3_1  ; 连续SK3
ANDNOT SK3_3  ; 寸动SK3
OUT 61.12  ; 单次
; rung 23
LD SK3_1  ; 连续SK3
ANDNOT SK3_2  ; 单次SK3
ANDNOT SK3_3  ; 寸动SK3
OUT 61.13  ; 连续
; rung 24
LD SK3_3  ; 寸动SK3
ANDNOT SK3_1  ; 连续SK3
ANDNOT SK3_2  ; 单次SK3
OUT 61.14  ; 寸动
; rung 25
LDNOT SP26  ; 离制压力
LD 61.15  ; 离制压力
ANDNOT SB26  ; 故障复位
ORLD
OUT 61.15  ; 离制压力
; rung 26
LD 0.00  ; 右前按钮站闭点并
AND 0.04  ; 左后按钮站闭点并
OUT 62.01  ; 闭点并
; rung 27
LD 0.01  ; 右前按钮站闭点串
AND 0.05  ; 左后按钮站闭点串
OUT 62.02  ; 闭点串
; rung 28
LD 0.02  ; 右前按钮站开点串
AND 0.06  ; 左后按钮站开点串
OUT 62.03  ; 开点串
; rung 29
LD SK2_2  ; 选择行程
AND HL5  ; 润滑正常
ANDNOT 61.15  ; 离制压力
ANDNOT SK6  ; 数据编辑
AND 33.04  ; 液保与行程连锁
AND KA9  ; 安全栓
AND 41.10  ; 装模高度与行程联锁
AND 52.04  ; 工作台落下夹紧
AND 37.02  ; 故障复位
OUT 62.04  ; 开动条件
; rung 30
LD 61.12  ; 单次
OR 61.13  ; 连续
LD 34.02  ; 气垫压力正常
OR SQ2  ; 气垫落到底
ANDLD
LDNOT 63.11  ; 计数到
AND 63.13  ; 产品计数通/断
ORNOT 63.13  ; 产品计数通/断
OR CLSA_3  ; 单次返回180-330
ANDLD
AND 62.04  ; 开动条件
OUT 62.05  ; 单连条件
; rung 31
LD XS13  ; 右前移动按钮站插�
OR XS15  ; 左后移动按钮站插�
AND 62.05  ; 单连条件
AND HL1  ; 主电机运行
AND XS13  ; 右前移动按钮站插�
AND XS15  ; 左后移动按钮站插�
OUT HL15_16  ; 移动按钮站插入

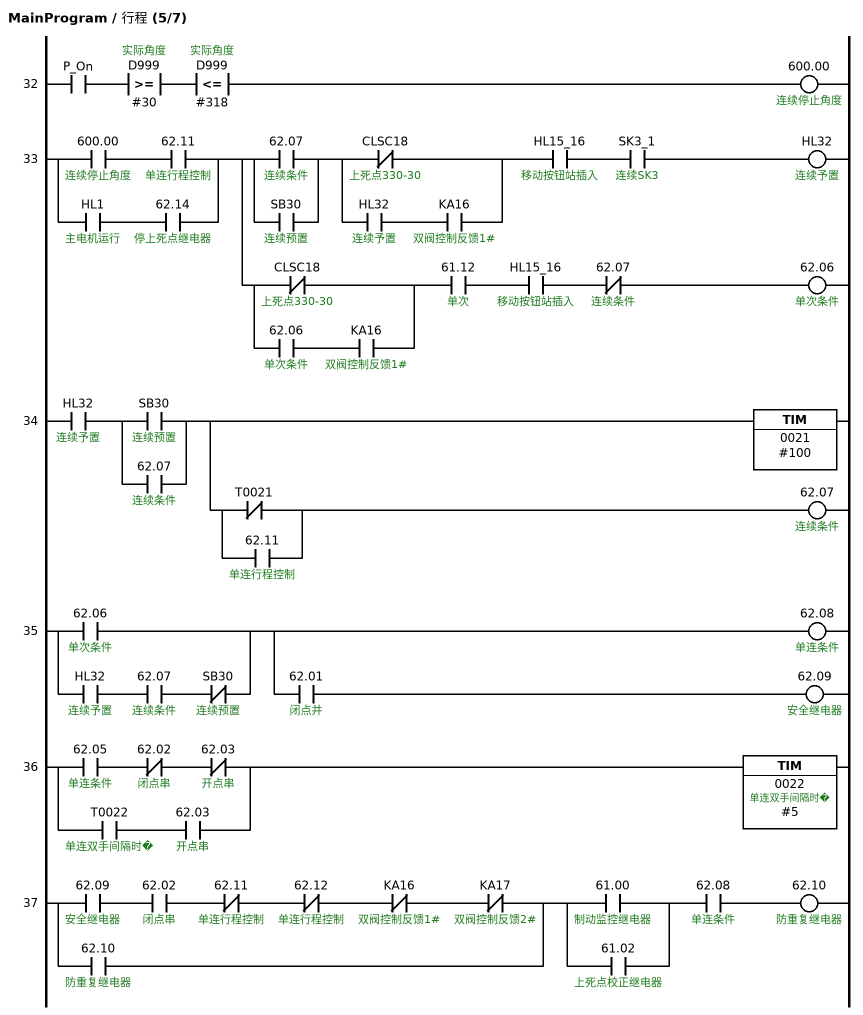
; rung 32
LD P_On
AND>=(325) D999 #30  ; 实际角度
AND<=(315) D999 #318  ; 实际角度
OUT 600.00  ; 连续停止角度
; rung 33
LD 600.00  ; 连续停止角度
AND 62.11  ; 单连行程控制
LD HL1  ; 主电机运行
AND 62.14  ; 停上死点继电器
ORLD
OUT TR0
LD 62.07  ; 连续条件
OR SB30  ; 连续预置
ANDLD
LDNOT CLSC18  ; 上死点330-30
LD HL32  ; 连续予置
AND KA16  ; 双阀控制反馈1#
ORLD
ANDLD
AND HL15_16  ; 移动按钮站插入
AND SK3_1  ; 连续SK3
OUT HL32  ; 连续予置
LD TR0
LDNOT CLSC18  ; 上死点330-30
LD 62.06  ; 单次条件
AND KA16  ; 双阀控制反馈1#
ORLD
ANDLD
AND 61.12  ; 单次
AND HL15_16  ; 移动按钮站插入
ANDNOT 62.07  ; 连续条件
OUT 62.06  ; 单次条件
; rung 34
LD HL32  ; 连续予置
LD SB30  ; 连续预置
OR 62.07  ; 连续条件
ANDLD
TIM 0021 #100
LDNOT T0021
OR 62.11  ; 单连行程控制
ANDLD
OUT 62.07  ; 连续条件
; rung 35
LD 62.06  ; 单次条件
LD HL32  ; 连续予置
AND 62.07  ; 连续条件
ANDNOT SB30  ; 连续预置
ORLD
OUT 62.08  ; 单连条件
AND 62.01  ; 闭点并
OUT 62.09  ; 安全继电器
; rung 36
LD 62.05  ; 单连条件
ANDNOT 62.02  ; 闭点串
ANDNOT 62.03  ; 开点串
LD T0022  ; 单连双手间隔时�
AND 62.03  ; 开点串
ORLD
TIM 0022 #5  ; 单连双手间隔时�
; rung 37
LD 62.09  ; 安全继电器
AND 62.02  ; 闭点串
ANDNOT 62.11  ; 单连行程控制
ANDNOT 62.12  ; 单连行程控制
ANDNOT KA16  ; 双阀控制反馈1#
ANDNOT KA17  ; 双阀控制反馈2#
OR 62.10  ; 防重复继电器
LD 61.00  ; 制动监控继电器
OR 61.02  ; 上死点校正继电器
ANDLD
AND 62.08  ; 单连条件
OUT 62.10  ; 防重复继电器

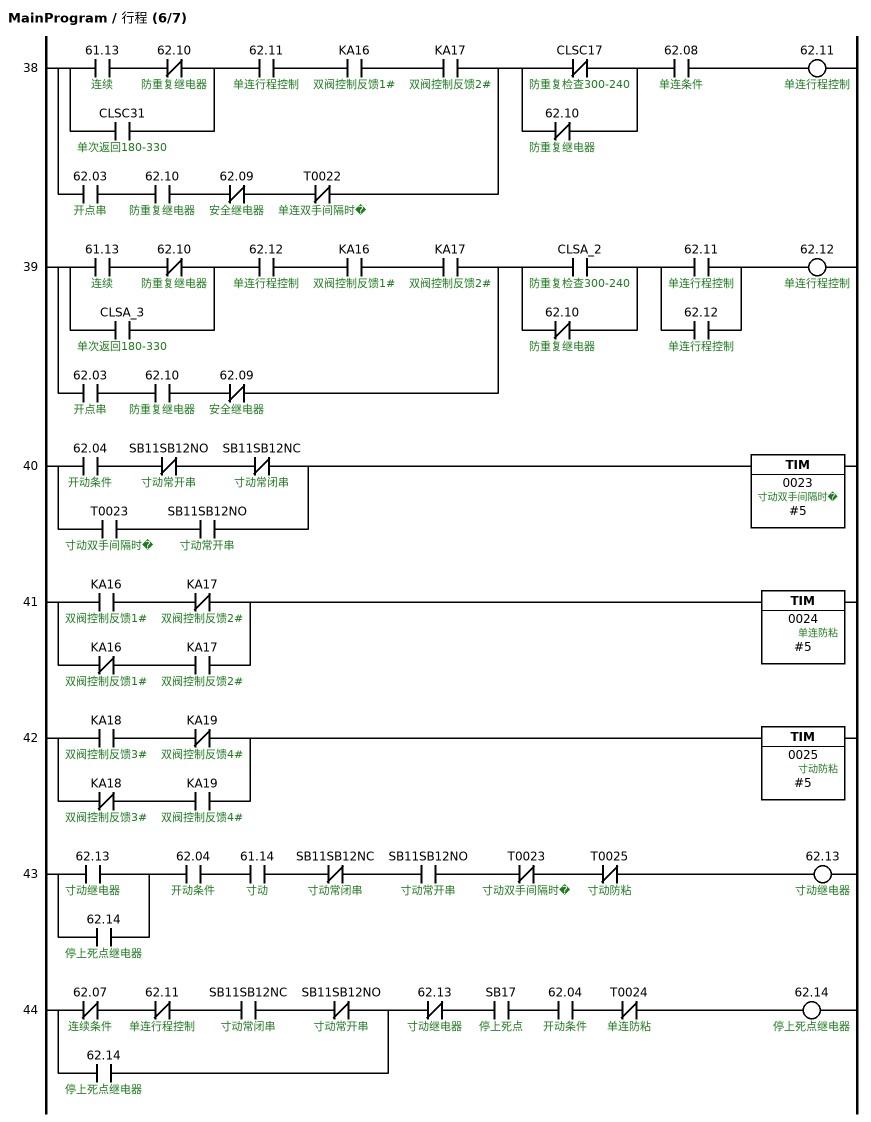
; rung 38
LD 61.13  ; 连续
ANDNOT 62.10  ; 防重复继电器
OR CLSC31  ; 单次返回180-330
AND 62.11  ; 单连行程控制
AND KA16  ; 双阀控制反馈1#
AND KA17  ; 双阀控制反馈2#
LD 62.03  ; 开点串
AND 62.10  ; 防重复继电器
ANDNOT 62.09  ; 安全继电器
ANDNOT T0022  ; 单连双手间隔时�
ORLD
LDNOT CLSC17  ; 防重复检查300-240
ORNOT 62.10  ; 防重复继电器
ANDLD
AND 62.08  ; 单连条件
OUT 62.11  ; 单连行程控制
; rung 39
LD 61.13  ; 连续
ANDNOT 62.10  ; 防重复继电器
OR CLSA_3  ; 单次返回180-330
AND 62.12  ; 单连行程控制
AND KA16  ; 双阀控制反馈1#
AND KA17  ; 双阀控制反馈2#
LD 62.03  ; 开点串
AND 62.10  ; 防重复继电器
ANDNOT 62.09  ; 安全继电器
ORLD
LD CLSA_2  ; 防重复检查300-240
ORNOT 62.10  ; 防重复继电器
ANDLD
LD 62.11  ; 单连行程控制
OR 62.12  ; 单连行程控制
ANDLD
OUT 62.12  ; 单连行程控制
; rung 40
LD 62.04  ; 开动条件
ANDNOT SB11SB12NO  ; 寸动常开串
ANDNOT SB11SB12NC  ; 寸动常闭串
LD T0023  ; 寸动双手间隔时�
AND SB11SB12NO  ; 寸动常开串
ORLD
TIM 0023 #5  ; 寸动双手间隔时�
; rung 41
LD KA16  ; 双阀控制反馈1#
ANDNOT KA17  ; 双阀控制反馈2#
LDNOT KA16  ; 双阀控制反馈1#
AND KA17  ; 双阀控制反馈2#
ORLD
TIM 0024 #5  ; 单连防粘
; rung 42
LD KA18  ; 双阀控制反馈3#
ANDNOT KA19  ; 双阀控制反馈4#
LDNOT KA18  ; 双阀控制反馈3#
AND KA19  ; 双阀控制反馈4#
ORLD
TIM 0025 #5  ; 寸动防粘
; rung 43
LD 62.13  ; 寸动继电器
OR 62.14  ; 停上死点继电器
AND 62.04  ; 开动条件
AND 61.14  ; 寸动
ANDNOT SB11SB12NC  ; 寸动常闭串
AND SB11SB12NO  ; 寸动常开串
ANDNOT T0023  ; 寸动双手间隔时�
ANDNOT T0025  ; 寸动防粘
OUT 62.13  ; 寸动继电器
; rung 44
LDNOT 62.07  ; 连续条件
ANDNOT 62.11  ; 单连行程控制
AND SB11SB12NC  ; 寸动常闭串
ANDNOT SB11SB12NO  ; 寸动常开串
OR 62.14  ; 停上死点继电器
ANDNOT 62.13  ; 寸动继电器
AND SB17  ; 停上死点
AND 62.04  ; 开动条件
ANDNOT T0024  ; 单连防粘
OUT 62.14  ; 停上死点继电器

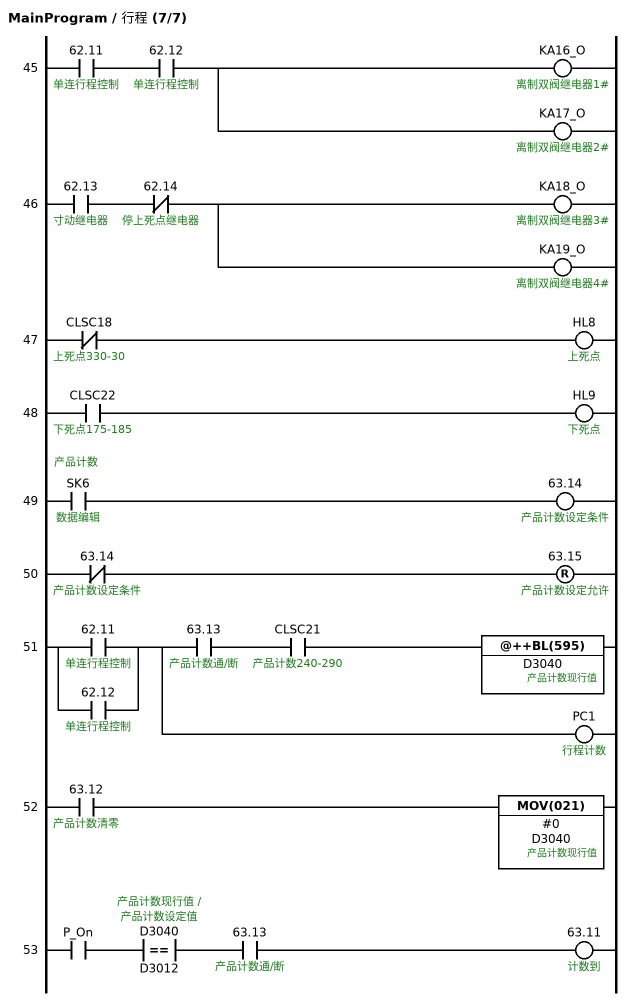
; rung 45
LD 62.11  ; 单连行程控制
AND 62.12  ; 单连行程控制
OUT KA16_O  ; 离制双阀继电器1#
OUT KA17_O  ; 离制双阀继电器2#
; rung 46
LD 62.13  ; 寸动继电器
ANDNOT 62.14  ; 停上死点继电器
OUT KA18_O  ; 离制双阀继电器3#
OUT KA19_O  ; 离制双阀继电器4#
; rung 47
LDNOT CLSC18  ; 上死点330-30
OUT HL8  ; 上死点
; rung 48
LD CLSC22  ; 下死点175-185
OUT HL9  ; 下死点
; rung 49: 产品计数
LD SK6  ; 数据编辑
OUT 63.14  ; 产品计数设定条件
; rung 50
LDNOT 63.14  ; 产品计数设定条件
RSET 63.15  ; 产品计数设定允许
; rung 51
LD 62.11  ; 单连行程控制
OR 62.12  ; 单连行程控制
OUT TR0
AND 63.13  ; 产品计数通/断
AND CLSC21  ; 产品计数240-290
@++BL(595) D3040  ; 产品计数现行值
LD TR0
OUT PC1  ; 行程计数
; rung 52
LD 63.12  ; 产品计数清零
MOV(021) #0 D3040  ; 产品计数现行值
; rung 53
LD P_On
AND=L(301) D3040 D3012  ; 产品计数现行值, 产品计数设定值
AND 63.13  ; 产品计数通/断
OUT 63.11  ; 计数到

### Section 滑块调整

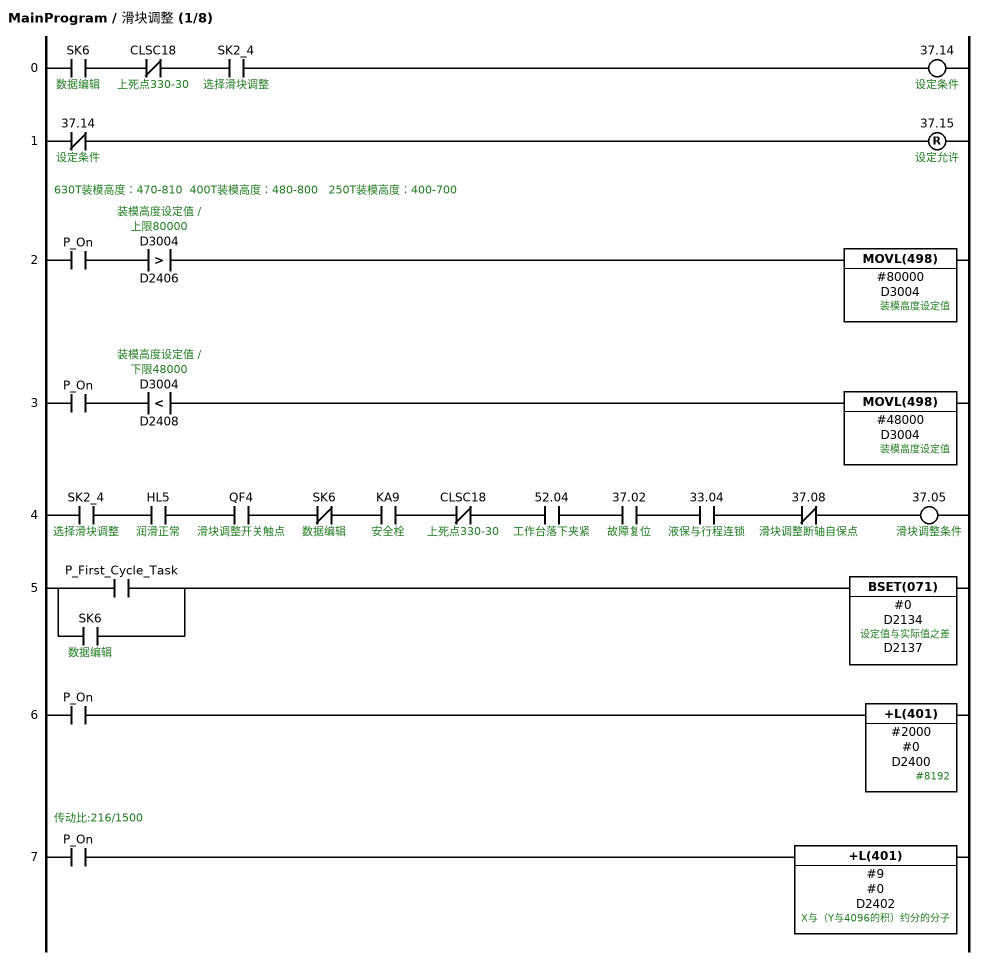
; rung 0
LD SK6  ; 数据编辑
ANDNOT CLSC18  ; 上死点330-30
AND SK2_4  ; 选择滑块调整
OUT 37.14  ; 设定条件
; rung 1
LDNOT 37.14  ; 设定条件
RSET 37.15  ; 设定允许
; rung 2: 630T装模高度：470-810  400T装模高度：480-800   250T装模高度：400-700
LD P_On
AND>L(321) D3004 D2406  ; 装模高度设定值, 上限80000
MOVL(498) #80000 D3004  ; 装模高度设定值
; rung 3
LD P_On
AND<L(311) D3004 D2408  ; 装模高度设定值, 下限48000
MOVL(498) #48000 D3004  ; 装模高度设定值
; rung 4
LD SK2_4  ; 选择滑块调整
AND HL5  ; 润滑正常
AND QF4  ; 滑块调整开关触点
ANDNOT SK6  ; 数据编辑
AND KA9  ; 安全栓
ANDNOT CLSC18  ; 上死点330-30
AND 52.04  ; 工作台落下夹紧
AND 37.02  ; 故障复位
AND 33.04  ; 液保与行程连锁
ANDNOT 37.08  ; 滑块调整断轴自保点
OUT 37.05  ; 滑块调整条件
; rung 5
LD P_First_Cycle_Task
OR SK6  ; 数据编辑
BSET(071) #0 D2134 D2137  ; 设定值与实际值之差
; rung 6
LD P_On
+L(401) #2000 #0 D2400  ; #8192
; rung 7: 传动比:216/1500
LD P_On
+L(401) #9 #0 D2402  ; X与（Y与4096的积）约分的分子

